C03655=1128.432,274.072,-72.523,-178.249,10.168,149.556
C03656=1128.428,274.321,-72.554,-178.246,10.171,149.556
C03657=1128.424,274.569,-72.583,-178.243,10.173,149.556
C03658=1128.420,274.818,-72.613,-178.240,10.176,149.556
C03659=1128.416,275.065,-72.643,-178.237,10.179,149.556
C03660=1128.412,275.314,-72.672,-178.234,10.181,149.556
C03661=1128.407,275.562,-72.702,-178.231,10.184,149.556
C03662=1128.403,275.810,-72.733,-178.228,10.187,149.555
C03663=1128.399,276.058,-72.762,-178.225,10.189,149.555
C03664=1128.395,276.306,-72.792,-178.221,10.193,149.555
C03665=1128.390,276.554,-72.822,-178.218,10.195,149.555
C03666=1128.386,276.803,-72.852,-178.215,10.198,149.555
C03667=1128.382,277.050,-72.882,-178.212,10.201,149.555
C03668=1128.377,277.299,-72.912,-178.209,10.203,149.554
C03669=1128.374,277.547,-72.943,-178.205,10.207,149.554
C03670=1128.370,277.795,-72.972,-178.202,10.209,149.554
C03671=1128.365,278.043,-73.003,-178.199,10.212,149.554
C03672=1128.361,278.292,-73.032,-178.196,10.214,149.554
C03673=1128.357,278.539,-73.062,-178.192,10.218,149.554
C03674=1128.352,278.788,-73.092,-178.189,10.220,149.553
C03675=1128.348,279.036,-73.123,-178.186,10.223,149.553
C03676=1128.345,279.285,-73.152,-178.182,10.226,149.553
C03677=1128.340,279.532,-73.183,-178.179,10.229,149.553
C03678=1128.336,279.780,-73.213,-178.175,10.231,149.553
C03679=1128.332,279.994,-73.239,-178.172,10.234,149.552
C03680=1128.329,280.207,-73.265,-178.169,10.237,149.552
C03681=1128.325,280.421,-73.291,-178.166,10.239,149.552
C03682=1128.321,280.634,-73.318,-178.163,10.241,149.552
C03683=1128.318,280.848,-73.343,-178.161,10.244,149.552
C03684=1128.314,281.061,-73.370,-178.157,10.246,149.551
C03685=1128.310,281.275,-73.395,-178.154,10.249,149.551
C03686=1128.307,281.489,-73.422,-178.151,10.251,149.551
C03687=1128.303,281.736,-73.452,-178.148,10.254,149.551
C03688=1128.298,281.984,-73.483,-178.145,10.257,149.551
C03689=1128.294,282.233,-73.512,-178.142,10.258,149.550
C03690=1128.290,282.481,-73.543,-178.139,10.261,149.550
C03691=1128.286,282.729,-73.574,-178.136,10.264,149.550
C03692=1128.282,282.977,-73.604,-178.133,10.266,149.550
C03693=1128.277,283.225,-73.634,-178.130,10.269,149.550
C03694=1128.274,283.474,-73.665,-178.127,10.272,149.550
C03695=1128.269,283.722,-73.696,-178.123,10.274,149.549
C03696=1128.265,283.969,-73.726,-178.121,10.277,149.549
C03697=1128.260,284.217,-73.756,-178.117,10.279,149.549
C03698=1128.257,284.466,-73.787,-178.114,10.282,149.549
C03699=1128.253,284.714,-73.818,-178.112,10.284,149.549
C03700=1128.248,284.962,-73.848,-178.109,10.286,149.548
C03701=1128.244,285.209,-73.879,-178.106,10.289,149.548
C03702=1128.240,285.458,-73.909,-178.102,10.292,149.548
C03703=1128.235,285.706,-73.940,-178.099,10.294,149.548
C03704=1128.231,285.954,-73.970,-178.096,10.297,149.548
C03705=1128.227,286.203,-74.001,-178.093,10.299,149.548
C03706=1128.223,286.451,-74.032,-178.090,10.302,149.547
C03707=1128.219,286.698,-74.062,-178.087,10.305,149.547
C03708=1128.215,286.947,-74.093,-178.084,10.307,149.547
C03709=1128.210,287.195,-74.124,-178.081,10.310,149.547
C03710=1128.206,287.443,-74.154,-178.078,10.312,149.547
C03711=1128.203,287.691,-74.186,-178.075,10.314,149.546
C03712=1128.198,287.939,-74.217,-178.072,10.317,149.546
C03713=1128.194,288.186,-74.247,-178.069,10.319,149.546
C03714=1128.190,288.435,-74.278,-178.066,10.322,149.546
C03715=1128.185,288.683,-74.309,-178.062,10.325,149.546
C03716=1128.181,288.931,-74.340,-178.059,10.327,149.546
C03717=1128.178,289.179,-74.370,-178.057,10.330,149.546
C03718=1128.173,289.427,-74.401,-178.053,10.333,149.545
C03719=1128.169,289.675,-74.433,-178.050,10.335,149.545
C03720=1128.165,289.923,-74.463,-178.048,10.337,149.545
C03721=1128.161,290.171,-74.494,-178.045,10.340,149.545
C03722=1128.157,290.419,-74.525,-178.041,10.342,149.545
C03723=1128.152,290.667,-74.556,-178.038,10.345,149.544
C03724=1128.148,290.915,-74.587,-178.035,10.347,149.544
C03725=1128.144,291.163,-74.618,-178.032,10.350,149.544
C03726=1128.141,291.412,-74.649,-178.029,10.353,149.544
C03727=1128.136,291.659,-74.680,-178.026,10.355,149.544
C03728=1128.132,291.907,-74.711,-178.022,10.358,149.543
C03729=1128.128,292.156,-74.742,-178.020,10.360,149.543
C03730=1128.123,292.403,-74.774,-178.017,10.363,149.543
C03731=1128.119,292.652,-74.805,-178.013,10.366,149.543
C03732=1128.115,292.900,-74.835,-178.011,10.368,149.543
C03733=1128.112,293.147,-74.867,-178.008,10.370,149.543
C03734=1128.107,293.395,-74.897,-178.005,10.373,149.543
C03735=1128.104,293.609,-74.924,-178.001,10.375,149.542
C03736=1128.100,293.822,-74.951,-177.999,10.377,149.542
C03737=1128.097,294.035,-74.978,-177.997,10.379,149.542
C03738=1128.093,294.249,-75.005,-177.994,10.382,149.542
C03739=1128.089,294.462,-75.032,-177.991,10.384,149.542
C03740=1128.086,294.676,-75.059,-177.989,10.386,149.542
C03741=1128.082,294.889,-75.086,-177.986,10.388,149.541
C03742=1128.079,295.103,-75.113,-177.983,10.390,149.541
C03743=1128.074,295.350,-75.143,-177.980,10.393,149.541
C03744=1128.070,295.599,-75.175,-177.977,10.395,149.541
C03745=1128.066,295.846,-75.206,-177.974,10.398,149.541
C03746=1128.062,296.095,-75.238,-177.971,10.401,149.541
C03747=1128.058,296.343,-75.270,-177.968,10.403,149.540
C03748=1128.054,296.591,-75.300,-177.965,10.406,149.540
C03749=1128.050,296.839,-75.332,-177.961,10.408,149.540
C03750=1128.045,297.086,-75.363,-177.958,10.411,149.540
C03751=1128.042,297.335,-75.395,-177.956,10.413,149.540
C03752=1128.037,297.582,-75.426,-177.953,10.416,149.540
C03753=1128.033,297.831,-75.458,-177.949,10.418,149.539
C03754=1128.029,298.078,-75.489,-177.947,10.421,149.539
C03755=1128.025,298.327,-75.520,-177.943,10.423,149.539
C03756=1128.021,298.575,-75.553,-177.940,10.426,149.539
C03757=1128.016,298.822,-75.584,-177.937,10.428,149.539
C03758=1128.013,299.070,-75.616,-177.934,10.431,149.538
C03759=1128.008,299.318,-75.647,-177.931,10.434,149.538
C03760=1128.004,299.566,-75.679,-177.928,10.436,149.538
C03761=1128.001,299.814,-75.710,-177.924,10.439,149.538
C03762=1127.996,300.062,-75.742,-177.921,10.441,149.538
C03763=1127.992,300.310,-75.773,-177.918,10.444,149.537
C03764=1127.987,300.558,-75.805,-177.915,10.446,149.537
C03765=1127.984,300.806,-75.837,-177.913,10.448,149.537
C03766=1127.980,301.054,-75.869,-177.909,10.451,149.537
C03767=1127.976,301.301,-75.900,-177.906,10.454,149.537
C03768=1127.971,301.550,-75.931,-177.903,10.456,149.537
C03769=1127.967,301.798,-75.964,-177.900,10.459,149.536
C03770=1127.963,302.046,-75.995,-177.897,10.461,149.536
C03771=1127.959,302.294,-76.027,-177.894,10.464,149.536
C03772=1127.955,302.541,-76.059,-177.890,10.466,149.536
C03773=1127.950,302.789,-76.091,-177.887,10.469,149.536
C03774=1127.947,303.037,-76.123,-177.884,10.472,149.535
C03775=1127.942,303.285,-76.154,-177.881,10.474,149.535
C03776=1127.939,303.533,-76.186,-177.878,10.477,149.535
C03777=1127.934,303.781,-76.219,-177.876,10.479,149.535
C03778=1127.930,304.029,-76.250,-177.872,10.481,149.535
C03779=1127.926,304.277,-76.282,-177.869,10.484,149.535
C03780=1127.922,304.525,-76.314,-177.866,10.486,149.534
C03781=1127.918,304.773,-76.346,-177.863,10.489,149.534
C03782=1127.914,305.020,-76.378,-177.860,10.492,149.534
C03783=1127.909,305.269,-76.410,-177.856,10.494,149.534
C03784=1127.906,305.517,-76.442,-177.853,10.497,149.534
C03785=1127.902,305.765,-76.474,-177.850,10.499,149.533
C03786=1127.897,306.012,-76.506,-177.847,10.502,149.533
C03787=1127.893,306.260,-76.538,-177.844,10.504,149.533
C03788=1127.889,306.508,-76.570,-177.841,10.507,149.533
C03789=1127.885,306.757,-76.602,-177.838,10.510,149.533
C03790=1127.881,307.004,-76.634,-177.835,10.512,149.533
C03791=1127.877,307.217,-76.661,-177.832,10.514,149.532
C03792=1127.874,307.431,-76.689,-177.830,10.516,149.532
C03793=1127.871,307.644,-76.717,-177.826,10.519,149.532
C03794=1127.866,307.857,-76.745,-177.824,10.521,149.532
C03795=1127.863,308.070,-76.772,-177.822,10.523,149.532
C03796=1127.860,308.283,-76.800,-177.818,10.525,149.532
C03797=1127.856,308.497,-76.828,-177.816,10.527,149.531
C03798=1127.853,308.710,-76.856,-177.813,10.530,149.531
C03799=1127.848,308.958,-76.888,-177.810,10.532,149.531
C03800=1127.845,309.205,-76.920,-177.808,10.534,149.531
C03801=1127.840,309.453,-76.953,-177.804,10.537,149.531
C03802=1127.836,309.701,-76.984,-177.801,10.539,149.531
C03803=1127.832,309.950,-77.017,-177.798,10.542,149.530
C03804=1127.829,310.197,-77.049,-177.795,10.544,149.530
C03805=1127.824,310.445,-77.082,-177.792,10.547,149.530
C03806=1127.820,310.692,-77.114,-177.788,10.549,149.530
C03807=1127.816,310.941,-77.147,-177.785,10.552,149.530
C03808=1127.812,311.189,-77.178,-177.782,10.555,149.530
C03809=1127.808,311.436,-77.212,-177.779,10.557,149.529
C03810=1127.804,311.684,-77.243,-177.776,10.560,149.529
C03811=1127.800,311.932,-77.277,-177.772,10.562,149.529
C03812=1127.796,312.179,-77.308,-177.770,10.565,149.529
C03813=1127.792,312.427,-77.341,-177.766,10.567,149.529
C03814=1127.787,312.676,-77.374,-177.763,10.570,149.529
C03815=1127.784,312.923,-77.406,-177.761,10.572,149.528
C03816=1127.779,313.171,-77.439,-177.757,10.574,149.528
C03817=1127.776,313.419,-77.471,-177.754,10.577,149.528
C03818=1127.771,313.667,-77.504,-177.751,10.580,149.528
C03819=1127.767,313.915,-77.537,-177.748,10.582,149.528
C03820=1127.764,314.163,-77.569,-177.745,10.585,149.527
C03821=1127.759,314.411,-77.602,-177.741,10.587,149.527
C03822=1127.754,314.658,-77.634,-177.739,10.590,149.527
C03823=1127.751,314.906,-77.666,-177.735,10.592,149.527
C03824=1127.747,315.153,-77.700,-177.732,10.595,149.526
C03825=1127.742,315.402,-77.732,-177.729,10.598,149.526
C03826=1127.739,315.649,-77.765,-177.726,10.600,149.526
C03827=1127.735,315.897,-77.798,-177.723,10.603,149.526
C03828=1127.730,316.145,-77.830,-177.719,10.605,149.526
C03829=1127.727,316.393,-77.863,-177.716,10.608,149.526
C03830=1127.723,316.640,-77.896,-177.713,10.611,149.525
C03831=1127.718,316.889,-77.928,-177.710,10.612,149.525
C03832=1127.714,317.136,-77.961,-177.707,10.615,149.525
C03833=1127.711,317.384,-77.994,-177.704,10.617,149.525
C03834=1127.707,317.632,-78.027,-177.701,10.620,149.525
C03835=1127.702,317.880,-78.060,-177.698,10.623,149.525
C03836=1127.698,318.128,-78.093,-177.695,10.625,149.524
C03837=1127.694,318.375,-78.126,-177.691,10.627,149.524
C03838=1127.691,318.623,-78.159,-177.688,10.630,149.524
C03839=1127.687,318.871,-78.192,-177.685,10.633,149.524
C03840=1127.682,319.118,-78.225,-177.682,10.635,149.524
C03841=1127.678,319.367,-78.257,-177.679,10.638,149.523
C03842=1127.674,319.614,-78.290,-177.675,10.640,149.523
C03843=1127.670,319.862,-78.323,-177.672,10.643,149.523
C03844=1127.667,320.110,-78.357,-177.669,10.646,149.523
C03845=1127.663,320.358,-78.390,-177.666,10.648,149.523
C03846=1127.659,320.606,-78.423,-177.663,10.651,149.523
C03847=1127.655,320.819,-78.452,-177.660,10.652,149.522
C03848=1127.652,321.032,-78.479,-177.658,10.654,149.522
C03849=1127.648,321.245,-78.508,-177.655,10.657,149.522
C03850=1127.645,321.458,-78.536,-177.652,10.659,149.522
C03851=1127.641,321.671,-78.565,-177.649,10.662,149.522
C03852=1127.638,321.884,-78.594,-177.647,10.663,149.521
C03853=1127.635,322.097,-78.622,-177.644,10.665,149.521
C03854=1127.631,322.310,-78.651,-177.641,10.668,149.521
C03855=1127.627,322.558,-78.684,-177.638,10.671,149.521
C03856=1127.623,322.805,-78.717,-177.635,10.673,149.521
C03857=1127.619,323.053,-78.750,-177.631,10.675,149.521
C03858=1127.614,323.301,-78.783,-177.629,10.677,149.520
C03859=1127.611,323.549,-78.817,-177.626,10.680,149.520
C03860=1127.607,323.796,-78.851,-177.623,10.682,149.520
C03861=1127.603,324.044,-78.884,-177.620,10.685,149.520
C03862=1127.599,324.292,-78.917,-177.616,10.688,149.520
C03863=1127.595,324.540,-78.950,-177.613,10.690,149.519
C03864=1127.591,324.787,-78.983,-177.610,10.693,149.519
C03865=1127.586,325.035,-79.016,-177.607,10.695,149.519
C03866=1127.583,325.283,-79.051,-177.603,10.698,149.519
C03867=1127.579,325.531,-79.084,-177.600,10.700,149.519
C03868=1127.575,325.778,-79.117,-177.597,10.703,149.519
C03869=1127.571,326.026,-79.150,-177.594,10.705,149.518
C03870=1127.567,326.273,-79.184,-177.590,10.708,149.518
C03871=1127.563,326.521,-79.217,-177.588,10.711,149.518
C03872=1127.559,326.769,-79.251,-177.584,10.713,149.518
C03873=1127.555,327.016,-79.284,-177.581,10.715,149.517
C03874=1127.551,327.264,-79.318,-177.578,10.718,149.517
C03875=1127.546,327.512,-79.351,-177.575,10.721,149.517
C03876=1127.543,327.760,-79.386,-177.571,10.723,149.517
C03877=1127.539,328.008,-79.419,-177.569,10.725,149.517
C03878=1127.535,328.255,-79.452,-177.566,10.728,149.517
C03879=1127.531,328.503,-79.486,-177.562,10.730,149.516
C03880=1127.527,328.750,-79.519,-177.559,10.733,149.516
C03881=1127.523,328.999,-79.552,-177.556,10.735,149.516
C03882=1127.519,329.246,-79.587,-177.553,10.738,149.516
C03883=1127.515,329.494,-79.620,-177.550,10.740,149.516
C03884=1127.511,329.741,-79.654,-177.547,10.743,149.515
C03885=1127.507,329.989,-79.688,-177.543,10.745,149.515
C03886=1127.503,330.237,-79.722,-177.540,10.748,149.515
C03887=1127.499,330.485,-79.755,-177.537,10.750,149.515
C03888=1127.495,330.732,-79.789,-177.534,10.753,149.515
C03889=1127.491,330.980,-79.823,-177.530,10.755,149.514
C03890=1127.487,331.227,-79.856,-177.527,10.758,149.514
C03891=1127.483,331.475,-79.890,-177.524,10.761,149.514
C03892=1127.479,331.723,-79.924,-177.521,10.763,149.514
C03893=1127.475,331.970,-79.958,-177.518,10.766,149.514
C03894=1127.471,332.218,-79.992,-177.514,10.768,149.513
C03895=1127.467,332.466,-80.026,-177.511,10.771,149.513
C03896=1127.464,332.713,-80.060,-177.508,10.773,149.513
C03897=1127.459,332.961,-80.093,-177.505,10.775,149.513
C03898=1127.455,333.209,-80.128,-177.502,10.777,149.513
C03899=1127.452,333.456,-80.162,-177.499,10.780,149.513
C03900=1127.447,333.704,-80.195,-177.496,10.783,149.512
C03901=1127.443,333.952,-80.230,-177.492,10.785,149.512
C03902=1127.440,334.199,-80.264,-177.489,10.788,149.512
C03903=1127.436,334.412,-80.293,-177.486,10.790,149.512
C03904=1127.433,334.626,-80.322,-177.483,10.792,149.512
C03905=1127.429,334.838,-80.352,-177.481,10.794,149.511
C03906=1127.426,335.051,-80.381,-177.478,10.796,149.511
C03907=1127.422,335.264,-80.410,-177.476,10.798,149.511
C03908=1127.420,335.477,-80.440,-177.472,10.801,149.511
C03909=1127.416,335.690,-80.469,-177.470,10.803,149.511
C03910=1127.412,335.903,-80.498,-177.467,10.805,149.511
C03911=1127.408,336.150,-80.532,-177.464,10.807,149.510
C03912=1127.405,336.398,-80.566,-177.461,10.810,149.510
C03913=1127.400,336.645,-80.601,-177.458,10.812,149.510
C03914=1127.397,336.893,-80.635,-177.454,10.815,149.510
C03915=1127.392,337.140,-80.670,-177.451,10.817,149.509
C03916=1127.389,337.389,-80.703,-177.448,10.820,149.509
C03917=1127.384,337.636,-80.738,-177.445,10.822,149.509
C03918=1127.380,337.883,-80.771,-177.442,10.825,149.509
C03919=1127.376,338.132,-80.806,-177.438,10.827,149.509
C03920=1127.373,338.379,-80.840,-177.435,10.830,149.509
C03921=1127.369,338.627,-80.875,-177.432,10.833,149.508
C03922=1127.365,338.874,-80.909,-177.429,10.835,149.508
C03923=1127.361,339.122,-80.944,-177.425,10.837,149.508
C03924=1127.357,339.369,-80.978,-177.422,10.840,149.508
C03925=1127.353,339.617,-81.012,-177.419,10.843,149.508
C03926=1127.348,339.865,-81.047,-177.416,10.845,149.507
C03927=1127.345,340.112,-81.081,-177.412,10.848,149.507
C03928=1127.341,340.360,-81.116,-177.409,10.850,149.507
C03929=1127.338,340.607,-81.150,-177.406,10.852,149.507
C03930=1127.333,340.854,-81.185,-177.404,10.854,149.507
C03931=1127.329,341.102,-81.219,-177.400,10.857,149.506
C03932=1127.325,341.350,-81.254,-177.397,10.859,149.506
C03933=1127.321,341.598,-81.288,-177.394,10.862,149.506
C03934=1127.317,341.845,-81.323,-177.390,10.864,149.506
C03935=1127.314,342.093,-81.357,-177.387,10.867,149.505
C03936=1127.309,342.340,-81.392,-177.384,10.870,149.505
C03937=1127.305,342.588,-81.427,-177.381,10.872,149.505
C03938=1127.302,342.835,-81.461,-177.377,10.874,149.505
C03939=1127.298,343.083,-81.496,-177.374,10.877,149.505
C03940=1127.293,343.330,-81.531,-177.371,10.879,149.505
C03941=1127.290,343.578,-81.565,-177.368,10.882,149.504
C03942=1127.286,343.825,-81.600,-177.365,10.885,149.504
C03943=1127.282,344.073,-81.635,-177.361,10.887,149.504
C03944=1127.278,344.320,-81.669,-177.358,10.890,149.504
C03945=1127.274,344.568,-81.704,-177.355,10.892,149.504
C03946=1127.270,344.816,-81.739,-177.351,10.894,149.503
C03947=1127.266,345.063,-81.774,-177.348,10.897,149.503
C03948=1127.262,345.311,-81.809,-177.345,10.900,149.503
C03949=1127.258,345.557,-81.843,-177.342,10.902,149.503
C03950=1127.254,345.806,-81.878,-177.338,10.905,149.503
C03951=1127.250,346.054,-81.913,-177.335,10.907,149.502
C03952=1127.246,346.301,-81.948,-177.332,10.910,149.502
C03953=1127.243,346.548,-81.983,-177.329,10.911,149.502
C03954=1127.239,346.795,-82.018,-177.326,10.914,149.502
C03955=1127.235,347.043,-82.053,-177.323,10.916,149.502
C03956=1127.231,347.291,-82.088,-177.320,10.919,149.501
C03957=1127.226,347.538,-82.123,-177.316,10.921,149.501
C03958=1127.223,347.786,-82.158,-177.313,10.924,149.501
C03959=1127.220,347.998,-82.188,-177.310,10.926,149.501
C03960=1127.216,348.211,-82.218,-177.307,10.928,149.501
C03961=1127.213,348.423,-82.248,-177.305,10.930,149.500
C03962=1127.210,348.637,-82.278,-177.302,10.933,149.500
C03963=1127.206,348.849,-82.309,-177.299,10.934,149.500
C03964=1127.203,349.062,-82.339,-177.296,10.937,149.500
C03965=1127.199,349.275,-82.369,-177.293,10.939,149.500
C03966=1127.197,349.488,-82.399,-177.291,10.941,149.499
C03967=1127.193,349.736,-82.434,-177.287,10.944,149.499
C03968=1127.188,349.983,-82.469,-177.284,10.946,149.499
C03969=1127.185,350.230,-82.504,-177.280,10.950,149.499
C03970=1127.181,350.478,-82.539,-177.276,10.952,149.498
C03971=1127.176,350.725,-82.574,-177.273,10.954,149.498
C03972=1127.173,350.973,-82.610,-177.269,10.957,149.498
C03973=1127.169,351.220,-82.645,-177.265,10.960,149.498
C03974=1127.165,351.468,-82.680,-177.262,10.962,149.497
C03975=1127.161,351.715,-82.715,-177.258,10.965,149.497
C03976=1127.157,351.963,-82.751,-177.254,10.968,149.497
C03977=1127.154,352.210,-82.787,-177.251,10.970,149.497
C03978=1127.150,352.458,-82.821,-177.248,10.973,149.497
C03979=1127.145,352.705,-82.857,-177.243,10.976,149.496
C03980=1127.142,352.952,-82.892,-177.240,10.978,149.496
C03981=1127.138,353.200,-82.928,-177.237,10.980,149.496
C03982=1127.134,353.448,-82.963,-177.233,10.983,149.495
C03983=1127.131,353.695,-82.999,-177.229,10.986,149.495
C03984=1127.126,353.942,-83.034,-177.226,10.988,149.495
C03985=1127.123,354.189,-83.069,-177.223,10.991,149.495
C03986=1127.119,354.437,-83.104,-177.219,10.993,149.494
C03987=1127.114,354.685,-83.140,-177.215,10.996,149.494
C03988=1127.111,354.933,-83.176,-177.212,10.999,149.494
C03989=1127.106,355.180,-83.211,-177.208,11.001,149.494
C03990=1127.103,355.427,-83.247,-177.205,11.004,149.493
C03991=1127.099,355.675,-83.282,-177.201,11.006,149.493
C03992=1127.095,355.922,-83.318,-177.198,11.008,149.493
C03993=1127.092,356.170,-83.353,-177.194,11.011,149.493
C03994=1127.088,356.417,-83.390,-177.191,11.014,149.492
C03995=1127.084,356.664,-83.426,-177.187,11.016,149.492
C03996=1127.080,356.911,-83.461,-177.184,11.018,149.492
C03997=1127.076,357.159,-83.496,-177.180,11.021,149.491
C03998=1127.072,357.406,-83.532,-177.177,11.023,149.491
C03999=1127.069,357.654,-83.568,-177.173,11.025,149.491
C04000=1127.064,357.901,-83.604,-177.170,11.028,149.491
C04001=1127.061,358.149,-83.639,-177.166,11.031,149.490
C04002=1127.057,358.396,-83.676,-177.162,11.033,149.490
C04003=1127.054,358.643,-83.711,-177.159,11.036,149.490
C04004=1127.049,358.891,-83.747,-177.156,11.038,149.490
C04005=1127.046,359.139,-83.783,-177.153,11.041,149.489
C04006=1127.042,359.386,-83.818,-177.149,11.043,149.489
C04007=1127.038,359.632,-83.854,-177.145,11.045,149.489
C04008=1127.034,359.880,-83.890,-177.142,11.048,149.489
C04009=1127.030,360.128,-83.926,-177.139,11.050,149.488
C04010=1127.027,360.374,-83.962,-177.135,11.052,149.488
C04011=1127.022,360.622,-83.998,-177.132,11.055,149.488
C04012=1127.018,360.870,-84.034,-177.129,11.057,149.488
C04013=1127.015,361.117,-84.070,-177.125,11.060,149.487
C04014=1127.011,361.364,-84.106,-177.122,11.062,149.487
C04015=1127.008,361.577,-84.138,-177.119,11.064,149.487
C04016=1127.004,361.790,-84.168,-177.116,11.066,149.487
C04017=1127.001,362.002,-84.199,-177.113,11.068,149.486
C04018=1126.998,362.215,-84.230,-177.110,11.071,149.486
C04019=1126.995,362.428,-84.262,-177.107,11.072,149.486
C04020=1126.992,362.640,-84.293,-177.104,11.075,149.486
C04021=1126.988,362.853,-84.323,-177.101,11.076,149.485
C04022=1126.985,363.065,-84.354,-177.099,11.078,149.485
C04023=1126.981,363.312,-84.391,-177.095,11.081,149.485
C04024=1126.978,363.560,-84.426,-177.092,11.083,149.485
C04025=1126.973,363.807,-84.463,-177.089,11.086,149.485
C04026=1126.970,364.055,-84.499,-177.085,11.088,149.484
C04027=1126.966,364.302,-84.535,-177.082,11.090,149.484
C04028=1126.962,364.549,-84.571,-177.078,11.093,149.484
C04029=1126.958,364.796,-84.608,-177.075,11.095,149.483
C04030=1126.955,365.045,-84.644,-177.072,11.098,149.483
C04031=1126.951,365.292,-84.681,-177.069,11.100,149.483
C04032=1126.947,365.539,-84.717,-177.065,11.103,149.483
C04033=1126.943,365.786,-84.753,-177.062,11.104,149.482
C04034=1126.940,366.033,-84.789,-177.059,11.106,149.482
C04035=1126.936,366.281,-84.826,-177.056,11.109,149.482
C04036=1126.932,366.528,-84.862,-177.052,11.111,149.482
C04037=1126.928,366.775,-84.899,-177.049,11.114,149.482
C04038=1126.924,367.022,-84.935,-177.046,11.116,149.481
C04039=1126.920,367.270,-84.971,-177.042,11.119,149.481
C04040=1126.917,367.517,-85.007,-177.039,11.121,149.481
C04041=1126.913,367.764,-85.044,-177.036,11.123,149.481
C04042=1126.909,368.012,-85.081,-177.033,11.125,149.480
C04043=1126.905,368.259,-85.117,-177.030,11.128,149.480
C04044=1126.901,368.507,-85.154,-177.026,11.130,149.480
C04045=1126.898,368.753,-85.190,-177.023,11.132,149.480
C04046=1126.894,369.001,-85.227,-177.019,11.135,149.479
C04047=1126.890,369.248,-85.264,-177.017,11.137,149.479
C04048=1126.886,369.495,-85.299,-177.014,11.139,149.479
C04049=1126.882,369.743,-85.336,-177.010,11.142,149.479
C04050=1126.879,369.990,-85.373,-177.007,11.144,149.479
C04051=1126.875,370.237,-85.410,-177.004,11.147,149.478
C04052=1126.871,370.485,-85.446,-177.001,11.148,149.478
C04053=1126.867,370.732,-85.483,-176.998,11.151,149.478
C04054=1126.864,370.979,-85.520,-176.994,11.153,149.478
C04055=1126.860,371.226,-85.557,-176.991,11.156,149.478
C04056=1126.856,371.474,-85.594,-176.989,11.158,149.477
C04057=1126.853,371.721,-85.630,-176.985,11.160,149.477
C04058=1126.849,371.968,-85.667,-176.982,11.163,149.477
C04059=1126.845,372.215,-85.704,-176.979,11.165,149.477
C04060=1126.841,372.463,-85.741,-176.976,11.168,149.477
C04061=1126.838,372.710,-85.777,-176.973,11.169,149.476
C04062=1126.834,372.957,-85.814,-176.970,11.172,149.476
C04063=1126.829,373.204,-85.851,-176.966,11.174,149.476
C04064=1126.825,373.451,-85.888,-176.963,11.177,149.476
C04065=1126.823,373.699,-85.924,-176.961,11.179,149.476
C04066=1126.819,373.946,-85.961,-176.957,11.181,149.475
C04067=1126.814,374.193,-85.998,-176.954,11.184,149.475
C04068=1126.810,374.440,-86.035,-176.951,11.185,149.475
C04069=1126.807,374.688,-86.072,-176.949,11.188,149.475
C04070=1126.804,374.935,-86.109,-176.945,11.191,149.475
C04071=1126.800,375.148,-86.141,-176.943,11.192,149.475
C04072=1126.797,375.360,-86.172,-176.940,11.194,149.474
C04073=1126.793,375.573,-86.205,-176.938,11.196,149.474
C04074=1126.790,375.785,-86.236,-176.935,11.199,149.474
C04075=1126.788,375.997,-86.268,-176.932,11.201,149.474
C04076=1126.784,376.210,-86.300,-176.930,11.203,149.474
C04077=1126.781,376.422,-86.332,-176.928,11.205,149.474
C04078=1126.777,376.634,-86.363,-176.925,11.206,149.474
C04079=1126.774,376.882,-86.400,-176.922,11.209,149.473
C04080=1126.770,377.129,-86.438,-176.919,11.212,149.473
C04081=1126.766,377.376,-86.474,-176.916,11.213,149.473
C04082=1126.763,377.624,-86.512,-176.913,11.216,149.473
C04083=1126.759,377.870,-86.549,-176.910,11.219,149.473
C04084=1126.755,378.117,-86.586,-176.907,11.220,149.473
C04085=1126.751,378.365,-86.623,-176.904,11.223,149.473
C04086=1126.748,378.612,-86.661,-176.901,11.226,149.472
C04087=1126.743,378.859,-86.698,-176.899,11.228,149.472
C04088=1126.740,379.107,-86.735,-176.895,11.230,149.472
C04089=1126.736,379.354,-86.773,-176.892,11.233,149.472
C04090=1126.732,379.601,-86.809,-176.890,11.235,149.472
C04091=1126.729,379.848,-86.847,-176.887,11.237,149.472
C04092=1126.725,380.095,-86.884,-176.884,11.240,149.472
C04093=1126.721,380.342,-86.921,-176.881,11.242,149.472
C04094=1126.717,380.590,-86.959,-176.878,11.245,149.472
C04095=1126.713,380.837,-86.996,-176.875,11.247,149.472
C04096=1126.710,381.084,-87.034,-176.873,11.249,149.471
C04097=1126.706,381.331,-87.071,-176.870,11.252,149.471
C04098=1126.702,381.578,-87.108,-176.867,11.254,149.471
C04099=1126.699,381.826,-87.146,-176.864,11.257,149.471
C04100=1126.695,382.072,-87.183,-176.862,11.259,149.471
C04101=1126.692,382.320,-87.220,-176.859,11.261,149.471
C04102=1126.688,382.567,-87.258,-176.856,11.264,149.471
C04103=1126.684,382.813,-87.295,-176.853,11.267,149.471
C04104=1126.680,383.061,-87.333,-176.851,11.269,149.471
C04105=1126.677,383.308,-87.370,-176.847,11.271,149.471
C04106=1126.673,383.556,-87.407,-176.846,11.274,149.471
C04107=1126.669,383.803,-87.446,-176.844,11.275,149.471
C04108=1126.665,384.049,-87.483,-176.842,11.277,149.471
C04109=1126.661,384.297,-87.520,-176.841,11.279,149.471
C04110=1126.658,384.544,-87.558,-176.839,11.281,149.471
C04111=1126.654,384.791,-87.596,-176.838,11.283,149.471
C04112=1126.650,385.038,-87.633,-176.836,11.284,149.471
C04113=1126.647,385.285,-87.671,-176.835,11.287,149.471
C04114=1126.643,385.532,-87.708,-176.833,11.288,149.471
C04115=1126.639,385.780,-87.746,-176.831,11.291,149.472
C04116=1126.635,386.027,-87.784,-176.830,11.292,149.472
C04117=1126.632,386.274,-87.822,-176.828,11.295,149.472
C04118=1126.628,386.521,-87.859,-176.827,11.296,149.472
C04119=1126.625,386.768,-87.896,-176.825,11.299,149.472
C04120=1126.621,387.015,-87.934,-176.824,11.300,149.472
C04121=1126.617,387.262,-87.972,-176.822,11.303,149.472
C04122=1126.613,387.510,-88.009,-176.821,11.304,149.473
C04123=1126.609,387.756,-88.047,-176.820,11.307,149.473
C04124=1126.606,388.004,-88.085,-176.818,11.309,149.473
C04125=1126.602,388.250,-88.123,-176.817,11.311,149.473
C04126=1126.599,388.498,-88.160,-176.816,11.313,149.473
C04127=1126.595,388.710,-88.192,-176.815,11.315,149.474
C04128=1126.592,388.923,-88.225,-176.813,11.317,149.474
C04129=1126.589,389.135,-88.257,-176.812,11.319,149.474
C04130=1126.586,389.347,-88.289,-176.811,11.321,149.474
C04131=1126.582,389.560,-88.322,-176.810,11.322,149.474
C04132=1126.580,389.772,-88.354,-176.809,11.324,149.475
C04133=1126.577,389.985,-88.387,-176.808,11.326,149.475
C04134=1126.573,390.197,-88.420,-176.806,11.329,149.475
C04135=1126.569,390.443,-88.457,-176.806,11.331,149.475
C04136=1126.566,390.691,-88.495,-176.804,11.333,149.476
C04137=1126.562,390.937,-88.533,-176.803,11.335,149.476
C04138=1126.558,391.185,-88.571,-176.802,11.338,149.476
C04139=1126.555,391.431,-88.609,-176.800,11.341,149.477
C04140=1126.551,391.679,-88.647,-176.799,11.342,149.477
C04141=1126.548,391.926,-88.685,-176.798,11.345,149.477
C04142=1126.544,392.173,-88.723,-176.797,11.347,149.477
C04143=1126.540,392.421,-88.760,-176.796,11.350,149.478
C04144=1126.536,392.667,-88.798,-176.795,11.353,149.478
C04145=1126.532,392.915,-88.836,-176.794,11.355,149.479
C04146=1126.529,393.162,-88.874,-176.793,11.358,149.479
C04147=1126.525,393.409,-88.912,-176.792,11.360,149.479
C04148=1126.522,393.655,-88.949,-176.791,11.363,149.480
C04149=1126.518,393.903,-88.988,-176.789,11.365,149.480
C04150=1126.514,394.150,-89.025,-176.789,11.367,149.481
C04151=1126.511,394.397,-89.063,-176.787,11.370,149.481
C04152=1126.507,394.644,-89.102,-176.786,11.373,149.481
C04153=1126.503,394.891,-89.139,-176.786,11.375,149.482
C04154=1126.500,395.138,-89.177,-176.785,11.378,149.482
C04155=1126.495,395.385,-89.216,-176.784,11.381,149.483
C04156=1126.492,395.632,-89.253,-176.782,11.384,149.483
C04157=1126.488,395.879,-89.291,-176.782,11.386,149.484
C04158=1126.484,396.127,-89.330,-176.780,11.389,149.484
C04159=1126.481,396.374,-89.368,-176.780,11.393,149.485
C04160=1126.477,396.620,-89.405,-176.779,11.395,149.485
C04161=1126.474,396.868,-89.444,-176.778,11.398,149.486
C04162=1126.470,397.114,-89.481,-176.777,11.401,149.486
C04163=1126.466,397.362,-89.520,-176.776,11.404,149.487
C04164=1126.463,397.609,-89.558,-176.776,11.406,149.488
C04165=1126.459,397.856,-89.595,-176.775,11.410,149.488
C04166=1126.455,398.103,-89.635,-176.774,11.413,149.489
C04167=1126.451,398.349,-89.672,-176.773,11.416,149.489
C04168=1126.448,398.597,-89.710,-176.772,11.419,149.490
C04169=1126.444,398.844,-89.749,-176.772,11.421,149.490
C04170=1126.441,399.091,-89.786,-176.771,11.425,149.491
C04171=1126.437,399.338,-89.825,-176.771,11.428,149.492
C04172=1126.433,399.585,-89.862,-176.769,11.431,149.492
C04173=1126.430,399.832,-89.900,-176.769,11.434,149.493
C04174=1126.426,400.079,-89.939,-176.768,11.438,149.494
C04175=1126.422,400.326,-89.977,-176.767,11.441,149.494
C04176=1126.418,400.573,-90.016,-176.767,11.444,149.495
C04177=1126.415,400.821,-90.053,-176.767,11.447,149.496
C04178=1126.411,401.068,-90.092,-176.766,11.450,149.496
C04179=1126.407,401.315,-90.130,-176.766,11.454,149.497
C04180=1126.405,401.561,-90.168,-176.765,11.457,149.498
C04181=1126.400,401.808,-90.206,-176.764,11.461,149.499
C04182=1126.397,402.056,-90.244,-176.764,11.464,149.500
C04183=1126.393,402.268,-90.277,-176.763,11.467,149.500
C04184=1126.390,402.480,-90.310,-176.763,11.470,149.501
C04185=1126.387,402.692,-90.343,-176.763,11.473,149.502
C04186=1126.384,402.904,-90.376,-176.762,11.476,149.502
C04187=1126.381,403.117,-90.409,-176.762,11.480,149.503
C04188=1126.377,403.329,-90.442,-176.762,11.482,149.504
C04189=1126.374,403.541,-90.475,-176.761,11.485,149.504
C04190=1126.371,403.753,-90.507,-176.761,11.488,149.505
C04191=1126.368,404.000,-90.546,-176.760,11.492,149.506
C04192=1126.364,404.247,-90.584,-176.760,11.495,149.507
C04193=1126.361,404.495,-90.623,-176.760,11.499,149.508
C04194=1126.357,404.741,-90.660,-176.759,11.503,149.508
C04195=1126.353,404.988,-90.699,-176.759,11.506,149.509
C04196=1126.350,405.236,-90.737,-176.759,11.510,149.510
C04197=1126.345,405.482,-90.776,-176.758,11.515,149.511
C04198=1126.343,405.729,-90.814,-176.758,11.518,149.512
C04199=1126.339,405.977,-90.853,-176.758,11.522,149.513
C04200=1126.335,406.223,-90.890,-176.758,11.526,149.514
C04201=1126.331,406.470,-90.930,-176.757,11.530,149.515
C04202=1126.328,406.717,-90.968,-176.758,11.534,149.516
C04203=1126.323,406.964,-91.006,-176.757,11.537,149.517
C04204=1126.320,407.211,-91.045,-176.757,11.541,149.518
C04205=1126.317,407.459,-91.083,-176.757,11.545,149.519
C04206=1126.313,407.705,-91.122,-176.757,11.550,149.520
C04207=1126.309,407.952,-91.160,-176.757,11.554,149.521
C04208=1126.305,408.200,-91.198,-176.757,11.558,149.522
C04209=1126.302,408.446,-91.237,-176.757,11.562,149.523
C04210=1126.299,408.694,-91.275,-176.757,11.566,149.524
C04211=1126.295,408.940,-91.314,-176.757,11.571,149.525
C04212=1126.291,409.187,-91.352,-176.757,11.575,149.526
C04213=1126.288,409.434,-91.392,-176.757,11.579,149.528
C04214=1126.284,409.681,-91.429,-176.757,11.583,149.529
C04215=1126.280,409.929,-91.468,-176.757,11.588,149.530
C04216=1126.277,410.175,-91.506,-176.757,11.592,149.531
C04217=1126.273,410.423,-91.545,-176.757,11.596,149.532
C04218=1126.269,410.669,-91.584,-176.757,11.601,149.533
C04219=1126.266,410.916,-91.622,-176.757,11.605,149.535
C04220=1126.262,411.163,-91.661,-176.757,11.610,149.536
C04221=1126.259,411.411,-91.699,-176.757,11.615,149.537
C04222=1126.255,411.657,-91.738,-176.758,11.619,149.538
C04223=1126.251,411.904,-91.776,-176.758,11.623,149.540
C04224=1126.248,412.151,-91.815,-176.758,11.629,149.541
C04225=1126.244,412.398,-91.854,-176.758,11.633,149.542
C04226=1126.240,412.646,-91.893,-176.758,11.638,149.543
C04227=1126.237,412.891,-91.931,-176.759,11.643,149.545
C04228=1126.233,413.139,-91.970,-176.760,11.647,149.546
C04229=1126.229,413.386,-92.009,-176.759,11.652,149.547
C04230=1126.226,413.633,-92.047,-176.760,11.657,149.549
C04231=1126.222,413.880,-92.086,-176.760,11.662,149.550
C04232=1126.219,414.126,-92.124,-176.761,11.666,149.551
C04233=1126.216,414.374,-92.163,-176.761,11.672,149.553
C04234=1126.213,414.621,-92.201,-176.762,11.676,149.554
C04235=1126.212,414.868,-92.240,-176.762,11.682,149.556
C04236=1126.212,415.115,-92.278,-176.763,11.687,149.557
C04237=1126.211,415.362,-92.316,-176.763,11.692,149.559
C04238=1126.211,415.609,-92.355,-176.764,11.697,149.560
C04239=1126.211,415.821,-92.387,-176.764,11.701,149.561
C04240=1126.213,416.033,-92.420,-176.765,11.705,149.563
C04241=1126.214,416.245,-92.453,-176.766,11.710,149.564
C04242=1126.216,416.457,-92.486,-176.766,11.714,149.565
C04243=1126.219,416.670,-92.517,-176.767,11.719,149.566
C04244=1126.221,416.881,-92.549,-176.767,11.723,149.568
C04245=1126.224,417.094,-92.582,-176.768,11.728,149.569
C04246=1126.228,417.305,-92.615,-176.769,11.732,149.571
C04247=1125.809,417.305,-92.678,-176.761,11.736,149.570
C04248=1125.806,417.093,-92.645,-176.761,11.732,149.569
C04249=1125.802,416.881,-92.613,-176.760,11.727,149.567
C04250=1125.799,416.668,-92.580,-176.760,11.723,149.566
C04251=1125.797,416.457,-92.548,-176.759,11.719,149.564
C04252=1125.795,416.245,-92.515,-176.758,11.714,149.563
C04253=1125.794,416.033,-92.482,-176.758,11.710,149.562
C04254=1125.792,415.821,-92.450,-176.757,11.705,149.561
C04255=1125.792,415.609,-92.417,-176.757,11.701,149.559
C04256=1125.792,415.362,-92.378,-176.756,11.695,149.558
C04257=1125.792,415.115,-92.340,-176.756,11.691,149.556
C04258=1125.793,414.868,-92.302,-176.755,11.685,149.555
C04259=1125.794,414.621,-92.264,-176.754,11.681,149.554
C04260=1125.797,414.373,-92.225,-176.755,11.676,149.552
C04261=1125.800,414.127,-92.186,-176.754,11.671,149.551
C04262=1125.803,413.880,-92.148,-176.754,11.666,149.549
C04263=1125.806,413.633,-92.109,-176.753,11.661,149.548
C04264=1125.810,413.386,-92.070,-176.753,11.656,149.547
C04265=1125.814,413.139,-92.032,-176.753,11.651,149.545
C04266=1125.817,412.892,-91.993,-176.753,11.646,149.544
C04267=1125.821,412.645,-91.955,-176.753,11.641,149.543
C04268=1125.824,412.398,-91.916,-176.752,11.637,149.541
C04269=1125.828,412.151,-91.877,-176.752,11.632,149.540
C04270=1125.832,411.904,-91.839,-176.752,11.627,149.539
C04271=1125.835,411.657,-91.800,-176.751,11.623,149.538
C04272=1125.839,411.410,-91.761,-176.752,11.618,149.536
C04273=1125.842,411.163,-91.723,-176.751,11.614,149.535
C04274=1125.847,410.916,-91.684,-176.752,11.609,149.534
C04275=1125.850,410.669,-91.645,-176.751,11.604,149.533
C04276=1125.853,410.422,-91.607,-176.751,11.600,149.532
C04277=1125.857,410.175,-91.568,-176.751,11.595,149.530
C04278=1125.861,409.929,-91.530,-176.751,11.591,149.529
C04279=1125.864,409.682,-91.491,-176.751,11.587,149.528
C04280=1125.868,409.434,-91.453,-176.751,11.582,149.527
C04281=1125.871,409.187,-91.414,-176.751,11.578,149.526
C04282=1125.876,408.940,-91.376,-176.751,11.574,149.525
C04283=1125.879,408.694,-91.337,-176.751,11.569,149.524
C04284=1125.883,408.446,-91.299,-176.751,11.565,149.523
C04285=1125.886,408.199,-91.259,-176.751,11.561,149.522
C04286=1125.890,407.953,-91.222,-176.751,11.557,149.520
C04287=1125.894,407.705,-91.183,-176.752,11.553,149.520
C04288=1125.897,407.458,-91.145,-176.752,11.549,149.519
C04289=1125.901,407.211,-91.106,-176.752,11.545,149.517
C04290=1125.904,406.965,-91.068,-176.752,11.541,149.516
C04291=1125.908,406.717,-91.029,-176.752,11.537,149.516
C04292=1125.911,406.470,-90.991,-176.753,11.532,149.514
C04293=1125.916,406.224,-90.952,-176.753,11.529,149.514
C04294=1125.920,405.976,-90.914,-176.753,11.525,149.512
C04295=1125.923,405.729,-90.876,-176.753,11.521,149.512
C04296=1125.926,405.482,-90.837,-176.754,11.517,149.511
C04297=1125.930,405.235,-90.799,-176.754,11.514,149.510
C04298=1125.934,404.988,-90.760,-176.755,11.509,149.509
C04299=1125.937,404.741,-90.722,-176.755,11.506,149.508
C04300=1125.941,404.494,-90.684,-176.755,11.502,149.507
C04301=1125.945,404.247,-90.646,-176.756,11.498,149.506
C04302=1125.948,404.000,-90.607,-176.756,11.495,149.505
C04303=1125.952,403.754,-90.569,-176.756,11.491,149.505
C04304=1125.955,403.541,-90.535,-176.757,11.488,149.504
C04305=1125.958,403.329,-90.503,-176.757,11.485,149.503
C04306=1125.962,403.116,-90.470,-176.758,11.481,149.502
C04307=1125.965,402.905,-90.437,-176.758,11.479,149.502
C04308=1125.968,402.692,-90.404,-176.758,11.475,149.501
C04309=1125.970,402.480,-90.371,-176.759,11.472,149.500
C04310=1125.974,402.268,-90.339,-176.759,11.470,149.500
C04311=1125.977,402.056,-90.306,-176.760,11.466,149.499
C04312=1125.981,401.809,-90.267,-176.760,11.463,149.498
C04313=1125.984,401.562,-90.229,-176.761,11.460,149.498
C04314=1125.988,401.315,-90.191,-176.761,11.456,149.497
C04315=1125.992,401.067,-90.153,-176.762,11.453,149.496
C04316=1125.995,400.821,-90.114,-176.763,11.449,149.495
C04317=1125.999,400.574,-90.076,-176.763,11.447,149.495
C04318=1126.002,400.326,-90.038,-176.764,11.443,149.494
C04319=1126.007,400.079,-90.000,-176.764,11.440,149.493
C04320=1126.010,399.832,-89.962,-176.765,11.437,149.493
C04321=1126.014,399.585,-89.924,-176.766,11.434,149.492
C04322=1126.017,399.339,-89.885,-176.767,11.430,149.491
C04323=1126.020,399.091,-89.847,-176.768,11.427,149.491
C04324=1126.025,398.845,-89.809,-176.769,11.424,149.490
C04325=1126.028,398.597,-89.771,-176.769,11.421,149.490
C04326=1126.032,398.350,-89.732,-176.769,11.418,149.489
C04327=1126.036,398.103,-89.695,-176.771,11.415,149.488
C04328=1126.039,397.856,-89.657,-176.771,11.412,149.488
C04329=1126.044,397.609,-89.619,-176.772,11.409,149.487
C04330=1126.046,397.362,-89.580,-176.773,11.406,149.487
C04331=1126.050,397.115,-89.542,-176.774,11.403,149.486
C04332=1126.054,396.868,-89.504,-176.775,11.400,149.486
C04333=1126.057,396.621,-89.466,-176.776,11.397,149.485
C04334=1126.062,396.374,-89.428,-176.777,11.394,149.484
C04335=1126.065,396.127,-89.390,-176.778,11.391,149.484
C04336=1126.068,395.879,-89.352,-176.779,11.388,149.483
C04337=1126.073,395.633,-89.314,-176.779,11.386,149.483
C04338=1126.076,395.385,-89.276,-176.780,11.383,149.483
C04339=1126.080,395.139,-89.238,-176.782,11.380,149.482
C04340=1126.084,394.891,-89.200,-176.783,11.377,149.482
C04341=1126.087,394.645,-89.162,-176.783,11.375,149.481
C04342=1126.091,394.397,-89.124,-176.785,11.372,149.481
C04343=1126.095,394.150,-89.086,-176.786,11.369,149.480
C04344=1126.098,393.903,-89.048,-176.787,11.367,149.480
C04345=1126.102,393.656,-89.010,-176.788,11.364,149.480
C04346=1126.106,393.409,-88.972,-176.789,11.361,149.479
C04347=1126.109,393.162,-88.934,-176.790,11.359,149.479
C04348=1126.113,392.915,-88.897,-176.791,11.356,149.478
C04349=1126.117,392.668,-88.858,-176.793,11.354,149.478
C04350=1126.121,392.421,-88.820,-176.793,11.352,149.478
C04351=1126.124,392.174,-88.782,-176.794,11.349,149.477
C04352=1126.128,391.927,-88.746,-176.796,11.346,149.477
C04353=1126.132,391.679,-88.707,-176.797,11.344,149.477
C04354=1126.135,391.432,-88.669,-176.798,11.341,149.476
C04355=1126.139,391.185,-88.632,-176.800,11.339,149.476
C04356=1126.142,390.938,-88.594,-176.801,11.337,149.476
C04357=1126.147,390.691,-88.555,-176.802,11.334,149.475
C04358=1126.150,390.444,-88.518,-176.804,11.331,149.475
C04359=1126.154,390.197,-88.480,-176.804,11.330,149.475
C04360=1126.157,389.985,-88.447,-176.806,11.328,149.475
C04361=1126.160,389.773,-88.415,-176.807,11.325,149.474
C04362=1126.163,389.560,-88.382,-176.808,11.323,149.474
C04363=1126.166,389.347,-88.350,-176.809,11.322,149.474
C04364=1126.169,389.135,-88.318,-176.810,11.320,149.474
C04365=1126.172,388.923,-88.285,-176.811,11.318,149.474
C04366=1126.176,388.711,-88.253,-176.813,11.316,149.473
C04367=1126.179,388.499,-88.221,-176.814,11.314,149.473
C04368=1126.183,388.252,-88.183,-176.815,11.312,149.473
C04369=1126.187,388.004,-88.145,-176.817,11.310,149.473
C04370=1126.190,387.757,-88.108,-176.818,11.307,149.473
C04371=1126.194,387.510,-88.070,-176.820,11.306,149.472
C04372=1126.197,387.263,-88.032,-176.821,11.303,149.472
C04373=1126.201,387.016,-87.995,-176.822,11.301,149.472
C04374=1126.205,386.769,-87.957,-176.824,11.299,149.472
C04375=1126.209,386.521,-87.919,-176.825,11.297,149.472
C04376=1126.212,386.275,-87.881,-176.827,11.295,149.472
C04377=1126.216,386.027,-87.844,-176.829,11.293,149.472
C04378=1126.220,385.780,-87.806,-176.830,11.291,149.471
C04379=1126.223,385.533,-87.769,-176.832,11.290,149.471
C04380=1126.227,385.286,-87.732,-176.834,11.287,149.471
C04381=1126.231,385.038,-87.693,-176.835,11.286,149.471
C04382=1126.235,384.792,-87.656,-176.837,11.283,149.471
C04383=1126.238,384.544,-87.618,-176.838,11.282,149.471
C04384=1126.242,384.297,-87.581,-176.840,11.279,149.471
C04385=1126.246,384.051,-87.543,-176.841,11.278,149.471
C04386=1126.249,383.803,-87.506,-176.843,11.276,149.471
C04387=1126.253,383.556,-87.468,-176.845,11.274,149.471
C04388=1126.256,383.309,-87.430,-176.847,11.272,149.471
C04389=1126.261,383.062,-87.393,-176.850,11.269,149.471
C04390=1126.264,382.814,-87.355,-176.852,11.267,149.471
C04391=1126.268,382.567,-87.318,-176.855,11.264,149.471
C04392=1126.272,382.320,-87.281,-176.858,11.262,149.471
C04393=1126.275,382.073,-87.243,-176.860,11.260,149.471
C04394=1126.279,381.826,-87.206,-176.863,11.257,149.471
C04395=1126.283,381.579,-87.168,-176.866,11.255,149.471
C04396=1126.287,381.332,-87.131,-176.869,11.253,149.471
C04397=1126.290,381.085,-87.093,-176.872,11.250,149.471
C04398=1126.294,380.837,-87.056,-176.874,11.248,149.471
C04399=1126.298,380.591,-87.019,-176.877,11.245,149.472
C04400=1126.301,380.343,-86.981,-176.880,11.242,149.472
C04401=1126.305,380.096,-86.944,-176.883,11.241,149.472
C04402=1126.309,379.849,-86.907,-176.886,11.238,149.472
C04403=1126.313,379.601,-86.870,-176.889,11.235,149.472
C04404=1126.316,379.354,-86.832,-176.891,11.233,149.472
C04405=1126.320,379.107,-86.795,-176.895,11.231,149.472
C04406=1126.324,378.860,-86.757,-176.898,11.228,149.472
C04407=1126.328,378.613,-86.721,-176.900,11.226,149.473
C04408=1126.332,378.366,-86.684,-176.903,11.224,149.473
C04409=1126.335,378.118,-86.646,-176.907,11.221,149.473
C04410=1126.339,377.871,-86.609,-176.909,11.219,149.473
C04411=1126.343,377.624,-86.572,-176.912,11.217,149.473
C04412=1126.346,377.377,-86.534,-176.915,11.214,149.473
C04413=1126.350,377.130,-86.498,-176.918,11.212,149.473
C04414=1126.354,376.883,-86.461,-176.921,11.210,149.473
C04415=1126.357,376.635,-86.424,-176.924,11.207,149.473
C04416=1126.361,376.422,-86.391,-176.927,11.205,149.474
C04417=1126.365,376.210,-86.360,-176.929,11.203,149.474
C04418=1126.367,375.998,-86.328,-176.931,11.201,149.474
C04419=1126.371,375.785,-86.296,-176.934,11.199,149.474
C04420=1126.374,375.573,-86.264,-176.937,11.197,149.474
C04421=1126.378,375.360,-86.233,-176.939,11.195,149.474
C04422=1126.380,375.148,-86.201,-176.942,11.193,149.475
C04423=1126.383,374.936,-86.169,-176.944,11.191,149.475
C04424=1126.387,374.689,-86.132,-176.948,11.189,149.475
C04425=1126.391,374.441,-86.095,-176.951,11.186,149.475
C04426=1126.395,374.194,-86.058,-176.954,11.184,149.475
C04427=1126.399,373.947,-86.021,-176.956,11.182,149.475
C04428=1126.402,373.700,-85.985,-176.960,11.179,149.476
C04429=1126.406,373.453,-85.948,-176.963,11.177,149.476
C04430=1126.410,373.205,-85.910,-176.966,11.174,149.476
C04431=1126.414,372.958,-85.874,-176.969,11.173,149.476
C04432=1126.417,372.711,-85.837,-176.972,11.170,149.476
C04433=1126.421,372.464,-85.800,-176.976,11.168,149.477
C04434=1126.425,372.216,-85.763,-176.978,11.165,149.477
C04435=1126.429,371.969,-85.726,-176.981,11.163,149.477
C04436=1126.432,371.722,-85.690,-176.984,11.161,149.477
C04437=1126.436,371.475,-85.653,-176.988,11.158,149.477
C04438=1126.440,371.227,-85.616,-176.991,11.156,149.477
C04439=1126.443,370.980,-85.580,-176.994,11.154,149.478
C04440=1126.447,370.733,-85.543,-176.997,11.151,149.478
C04441=1126.451,370.485,-85.506,-177.000,11.149,149.478
C04442=1126.455,370.238,-85.469,-177.004,11.147,149.478
C04443=1126.459,369.991,-85.433,-177.007,11.144,149.479
C04444=1126.463,369.743,-85.397,-177.010,11.142,149.479
C04445=1126.467,369.496,-85.360,-177.013,11.140,149.479
C04446=1126.470,369.249,-85.323,-177.016,11.137,149.479
C04447=1126.474,369.002,-85.286,-177.019,11.135,149.479
C04448=1126.478,368.755,-85.250,-177.023,11.132,149.480
C04449=1126.482,368.507,-85.213,-177.026,11.130,149.480
C04450=1126.486,368.260,-85.177,-177.029,11.128,149.480
C04451=1126.489,368.013,-85.141,-177.032,11.126,149.480
C04452=1126.493,367.765,-85.104,-177.035,11.123,149.481
C04453=1126.496,367.518,-85.067,-177.039,11.121,149.481
C04454=1126.501,367.270,-85.031,-177.042,11.118,149.481
C04455=1126.505,367.023,-84.994,-177.046,11.116,149.481
C04456=1126.508,366.776,-84.958,-177.048,11.115,149.482
C04457=1126.512,366.529,-84.921,-177.052,11.112,149.482
C04458=1126.516,366.281,-84.886,-177.055,11.110,149.482
C04459=1126.520,366.034,-84.849,-177.058,11.107,149.482
C04460=1126.524,365.787,-84.813,-177.062,11.105,149.482
C04461=1126.528,365.540,-84.776,-177.065,11.102,149.483
C04462=1126.531,365.293,-84.740,-177.068,11.100,149.483
C04463=1126.535,365.045,-84.704,-177.072,11.098,149.483
C04464=1126.538,364.797,-84.667,-177.075,11.095,149.483
C04465=1126.543,364.549,-84.631,-177.078,11.093,149.484
C04466=1126.546,364.303,-84.595,-177.081,11.091,149.484
C04467=1126.550,364.055,-84.558,-177.084,11.088,149.484
C04468=1126.554,363.808,-84.523,-177.088,11.086,149.484
C04469=1126.557,363.561,-84.486,-177.091,11.084,149.485
C04470=1126.561,363.313,-84.450,-177.095,11.081,149.485
C04471=1126.565,363.066,-84.414,-177.098,11.079,149.485
C04472=1126.568,362.853,-84.383,-177.101,11.077,149.485
C04473=1126.572,362.641,-84.352,-177.104,11.075,149.486
C04474=1126.575,362.428,-84.321,-177.107,11.073,149.486
C04475=1126.578,362.216,-84.290,-177.110,11.071,149.486
C04476=1126.582,362.004,-84.259,-177.112,11.069,149.486
C04477=1126.585,361.791,-84.228,-177.116,11.066,149.486
C04478=1126.588,361.578,-84.197,-177.118,11.064,149.487
C04479=1126.591,361.365,-84.166,-177.121,11.063,149.487
C04480=1126.595,361.118,-84.130,-177.124,11.060,149.487
C04481=1126.599,360.871,-84.094,-177.128,11.058,149.488
C04482=1126.602,360.623,-84.058,-177.131,11.056,149.488
C04483=1126.606,360.376,-84.022,-177.135,11.053,149.488
C04484=1126.611,360.129,-83.986,-177.138,11.051,149.488
C04485=1126.614,359.882,-83.950,-177.142,11.048,149.489
C04486=1126.618,359.634,-83.915,-177.145,11.045,149.489
C04487=1126.623,359.386,-83.879,-177.149,11.043,149.489
C04488=1126.626,359.139,-83.842,-177.152,11.040,149.489
C04489=1126.630,358.892,-83.807,-177.156,11.038,149.490
C04490=1126.633,358.644,-83.771,-177.159,11.036,149.490
C04491=1126.638,358.397,-83.735,-177.162,11.033,149.490
C04492=1126.641,358.150,-83.699,-177.166,11.031,149.490
C04493=1126.645,357.902,-83.663,-177.169,11.029,149.491
C04494=1126.648,357.655,-83.628,-177.173,11.026,149.491
C04495=1126.652,357.407,-83.592,-177.176,11.024,149.491
C04496=1126.656,357.159,-83.556,-177.179,11.021,149.491
C04497=1126.661,356.913,-83.521,-177.183,11.019,149.492
C04498=1126.664,356.665,-83.485,-177.187,11.016,149.492
C04499=1126.668,356.418,-83.450,-177.190,11.013,149.492
C04500=1126.672,356.170,-83.414,-177.194,11.011,149.492
C04501=1126.676,355.923,-83.377,-177.197,11.009,149.493
C04502=1126.679,355.675,-83.342,-177.201,11.006,149.493
C04503=1126.683,355.428,-83.306,-177.204,11.004,149.493
C04504=1126.687,355.181,-83.271,-177.208,11.001,149.493
C04505=1126.691,354.934,-83.236,-177.212,10.999,149.494
C04506=1126.695,354.686,-83.200,-177.215,10.996,149.494
C04507=1126.699,354.438,-83.165,-177.218,10.994,149.494
C04508=1126.702,354.190,-83.130,-177.222,10.991,149.494
C04509=1126.706,353.943,-83.094,-177.225,10.989,149.495
C04510=1126.711,353.696,-83.058,-177.229,10.986,149.495
C04511=1126.715,353.448,-83.023,-177.232,10.983,149.495
C04512=1126.718,353.201,-82.987,-177.236,10.981,149.496
C04513=1126.722,352.953,-82.952,-177.239,10.979,149.496
C04514=1126.726,352.707,-82.917,-177.243,10.976,149.496
C04515=1126.730,352.459,-82.881,-177.247,10.973,149.496
C04516=1126.734,352.211,-82.846,-177.250,10.971,149.497
C04517=1126.737,351.963,-82.811,-177.254,10.968,149.497
C04518=1126.741,351.716,-82.775,-177.258,10.965,149.497
C04519=1126.745,351.469,-82.740,-177.261,10.963,149.497
C04520=1126.749,351.221,-82.705,-177.264,10.960,149.498
C04521=1126.753,350.973,-82.670,-177.268,10.957,149.498
C04522=1126.757,350.727,-82.634,-177.272,10.955,149.498
C04523=1126.761,350.479,-82.599,-177.275,10.952,149.498
C04524=1126.765,350.231,-82.564,-177.279,10.949,149.499
C04525=1126.769,349.984,-82.528,-177.283,10.947,149.499
C04526=1126.772,349.737,-82.494,-177.286,10.944,149.499
C04527=1126.776,349.489,-82.459,-177.290,10.941,149.499
C04528=1126.779,349.276,-82.428,-177.292,10.939,149.500
C04529=1126.783,349.063,-82.398,-177.296,10.937,149.500
C04530=1126.787,348.851,-82.369,-177.298,10.935,149.500
C04531=1126.790,348.638,-82.338,-177.301,10.933,149.500
C04532=1126.793,348.425,-82.308,-177.304,10.931,149.500
C04533=1126.796,348.212,-82.278,-177.306,10.929,149.500
C04534=1126.800,347.999,-82.248,-177.310,10.926,149.501
C04535=1126.803,347.787,-82.218,-177.312,10.924,149.501
C04536=1126.807,347.540,-82.183,-177.315,10.922,149.501
C04537=1126.811,347.292,-82.147,-177.319,10.919,149.501
C04538=1126.815,347.044,-82.112,-177.322,10.917,149.501
C04539=1126.819,346.797,-82.078,-177.325,10.914,149.502
C04540=1126.822,346.549,-82.043,-177.329,10.912,149.502
C04541=1126.826,346.301,-82.008,-177.332,10.910,149.502
C04542=1126.831,346.055,-81.973,-177.335,10.907,149.502
C04543=1126.835,345.806,-81.938,-177.338,10.904,149.502
C04544=1126.838,345.560,-81.903,-177.341,10.902,149.503
C04545=1126.842,345.312,-81.868,-177.345,10.899,149.503
C04546=1126.846,345.064,-81.834,-177.347,10.898,149.503
C04547=1126.850,344.817,-81.798,-177.351,10.895,149.503
C04548=1126.854,344.569,-81.764,-177.354,10.893,149.504
C04549=1126.858,344.322,-81.730,-177.357,10.890,149.504
C04550=1126.862,344.074,-81.694,-177.360,10.888,149.504
C04551=1126.866,343.827,-81.660,-177.364,10.885,149.504
C04552=1126.870,343.579,-81.626,-177.367,10.883,149.504
C04553=1126.873,343.331,-81.590,-177.370,10.880,149.505
C04554=1126.878,343.084,-81.556,-177.373,10.878,149.505
C04555=1126.882,342.836,-81.521,-177.376,10.875,149.505
C04556=1126.886,342.589,-81.487,-177.380,10.872,149.505
C04557=1126.889,342.341,-81.451,-177.383,10.870,149.505
C04558=1126.894,342.094,-81.417,-177.386,10.868,149.506
C04559=1126.897,341.846,-81.383,-177.390,10.865,149.506
C04560=1126.902,341.599,-81.348,-177.393,10.863,149.506
C04561=1126.906,341.351,-81.313,-177.396,10.860,149.506
C04562=1126.910,341.103,-81.279,-177.399,10.857,149.506
C04563=1126.913,340.856,-81.244,-177.403,10.855,149.507
C04564=1126.917,340.609,-81.210,-177.406,10.852,149.507
C04565=1126.921,340.361,-81.175,-177.409,10.850,149.507
C04566=1126.926,340.113,-81.141,-177.412,10.847,149.507
C04567=1126.929,339.865,-81.106,-177.415,10.845,149.507
C04568=1126.933,339.618,-81.072,-177.418,10.843,149.508
C04569=1126.937,339.370,-81.038,-177.421,10.841,149.508
C04570=1126.941,339.123,-81.003,-177.425,10.838,149.508
C04571=1126.944,338.875,-80.969,-177.428,10.835,149.508
C04572=1126.949,338.628,-80.935,-177.431,10.833,149.508
C04573=1126.954,338.380,-80.900,-177.434,10.831,149.509
C04574=1126.957,338.132,-80.866,-177.438,10.828,149.509
C04575=1126.961,337.885,-80.831,-177.441,10.826,149.509
C04576=1126.965,337.637,-80.797,-177.444,10.823,149.509
C04577=1126.969,337.390,-80.763,-177.447,10.820,149.509
C04578=1126.972,337.142,-80.728,-177.450,10.818,149.510
C04579=1126.976,336.895,-80.695,-177.454,10.815,149.510
C04580=1126.980,336.646,-80.660,-177.457,10.813,149.510
C04581=1126.984,336.399,-80.627,-177.460,10.810,149.510
C04582=1126.989,336.152,-80.592,-177.463,10.808,149.510
C04583=1126.992,335.904,-80.558,-177.467,10.805,149.511
C04584=1126.996,335.691,-80.529,-177.469,10.803,149.511
C04585=1127.000,335.478,-80.499,-177.472,10.801,149.511
C04586=1127.002,335.265,-80.470,-177.475,10.799,149.511
C04587=1127.006,335.052,-80.441,-177.477,10.797,149.511
C04588=1127.009,334.840,-80.411,-177.480,10.794,149.511
C04589=1127.013,334.627,-80.382,-177.483,10.793,149.512
C04590=1127.016,334.414,-80.353,-177.486,10.790,149.512
C04591=1127.020,334.201,-80.323,-177.488,10.788,149.512
C04592=1127.024,333.953,-80.290,-177.492,10.786,149.512
C04593=1127.028,333.706,-80.256,-177.495,10.783,149.512
C04594=1127.032,333.458,-80.221,-177.498,10.781,149.512
C04595=1127.035,333.210,-80.187,-177.501,10.778,149.513
C04596=1127.040,332.963,-80.154,-177.505,10.776,149.513
C04597=1127.043,332.715,-80.119,-177.508,10.773,149.513
C04598=1127.047,332.467,-80.085,-177.511,10.770,149.513
C04599=1127.051,332.220,-80.052,-177.514,10.768,149.513
C04600=1127.055,331.972,-80.018,-177.517,10.766,149.514
C04601=1127.060,331.724,-79.984,-177.520,10.764,149.514
C04602=1127.063,331.477,-79.950,-177.523,10.761,149.514
C04603=1127.067,331.229,-79.916,-177.526,10.759,149.514
C04604=1127.072,330.981,-79.882,-177.529,10.756,149.514
C04605=1127.075,330.734,-79.848,-177.533,10.753,149.515
C04606=1127.079,330.485,-79.815,-177.536,10.751,149.515
C04607=1127.083,330.238,-79.781,-177.539,10.749,149.515
C04608=1127.087,329.991,-79.748,-177.542,10.746,149.515
C04609=1127.091,329.743,-79.713,-177.546,10.743,149.515
C04610=1127.095,329.495,-79.680,-177.549,10.741,149.516
C04611=1127.099,329.248,-79.646,-177.552,10.738,149.516
C04612=1127.103,329.000,-79.613,-177.555,10.736,149.516
C04613=1127.107,328.752,-79.580,-177.558,10.733,149.516
C04614=1127.111,328.504,-79.545,-177.562,10.731,149.516
C04615=1127.115,328.256,-79.512,-177.565,10.728,149.516
C04616=1127.119,328.009,-79.478,-177.568,10.726,149.517
C04617=1127.123,327.761,-79.445,-177.571,10.723,149.517
C04618=1127.127,327.514,-79.411,-177.574,10.720,149.517
C04619=1127.130,327.266,-79.377,-177.577,10.719,149.517
C04620=1127.135,327.018,-79.344,-177.580,10.716,149.518
C04621=1127.140,326.770,-79.310,-177.583,10.713,149.518
C04622=1127.143,326.523,-79.276,-177.587,10.711,149.518
C04623=1127.147,326.275,-79.243,-177.590,10.709,149.518
C04624=1127.151,326.027,-79.210,-177.593,10.706,149.518
C04625=1127.155,325.779,-79.177,-177.596,10.703,149.518
C04626=1127.159,325.532,-79.143,-177.599,10.701,149.519
C04627=1127.163,325.284,-79.110,-177.603,10.698,149.519
C04628=1127.167,325.037,-79.076,-177.606,10.696,149.519
C04629=1127.171,324.788,-79.043,-177.609,10.693,149.519
C04630=1127.175,324.540,-79.010,-177.612,10.691,149.519
C04631=1127.179,324.293,-78.976,-177.615,10.688,149.519
C04632=1127.183,324.046,-78.943,-177.619,10.686,149.520
C04633=1127.187,323.798,-78.909,-177.622,10.683,149.520
C04634=1127.191,323.550,-78.876,-177.625,10.680,149.520
C04635=1127.195,323.302,-78.843,-177.628,10.678,149.520
C04636=1127.199,323.054,-78.810,-177.631,10.675,149.521
C04637=1127.203,322.806,-78.777,-177.634,10.673,149.521
C04638=1127.207,322.559,-78.743,-177.637,10.671,149.521
C04639=1127.211,322.311,-78.710,-177.640,10.669,149.521
C04640=1127.215,322.098,-78.681,-177.643,10.666,149.521
C04641=1127.218,321.885,-78.653,-177.646,10.664,149.521
C04642=1127.221,321.672,-78.625,-177.649,10.661,149.522
C04643=1127.225,321.459,-78.596,-177.651,10.659,149.522
C04644=1127.228,321.246,-78.567,-177.654,10.658,149.522
C04645=1127.232,321.033,-78.540,-177.657,10.655,149.522
C04646=1127.235,320.820,-78.511,-177.660,10.653,149.522
C04647=1127.239,320.607,-78.482,-177.662,10.651,149.522
C04648=1127.243,320.359,-78.449,-177.665,10.649,149.523
C04649=1127.247,320.112,-78.415,-177.668,10.646,149.523
C04650=1127.251,319.864,-78.384,-177.671,10.644,149.523
C04651=1127.255,319.616,-78.350,-177.675,10.641,149.523
C04652=1127.259,319.368,-78.317,-177.678,10.638,149.523
C04653=1127.263,319.120,-78.284,-177.681,10.636,149.524
C04654=1127.267,318.873,-78.251,-177.684,10.633,149.524
C04655=1127.271,318.625,-78.218,-177.687,10.631,149.524
C04656=1127.275,318.378,-78.185,-177.691,10.628,149.524
C04657=1127.279,318.128,-78.152,-177.694,10.625,149.524
C04658=1127.283,317.881,-78.119,-177.697,10.623,149.524
C04659=1127.287,317.633,-78.086,-177.700,10.621,149.525
C04660=1127.290,317.386,-78.054,-177.703,10.618,149.525
C04661=1127.294,317.138,-78.020,-177.706,10.615,149.525
C04662=1127.299,316.890,-77.988,-177.710,10.613,149.525
C04663=1127.303,316.642,-77.955,-177.713,10.610,149.525
C04664=1127.306,316.394,-77.922,-177.715,10.609,149.526
C04665=1127.311,316.147,-77.890,-177.718,10.606,149.526
C04666=1127.315,315.899,-77.857,-177.722,10.603,149.526
C04667=1127.319,315.652,-77.824,-177.725,10.601,149.526
C04668=1127.323,315.403,-77.792,-177.728,10.598,149.526
C04669=1127.327,315.156,-77.759,-177.731,10.596,149.526
C04670=1127.331,314.908,-77.726,-177.734,10.593,149.527
C04671=1127.335,314.660,-77.694,-177.737,10.590,149.527
C04672=1127.339,314.412,-77.661,-177.741,10.588,149.527
C04673=1127.343,314.165,-77.628,-177.744,10.585,149.527
C04674=1127.347,313.916,-77.596,-177.747,10.583,149.527
C04675=1127.351,313.669,-77.563,-177.750,10.580,149.527
C04676=1127.355,313.420,-77.531,-177.753,10.578,149.528
C04677=1127.359,313.173,-77.498,-177.757,10.575,149.528
C04678=1127.364,312.924,-77.465,-177.760,10.572,149.528
C04679=1127.367,312.677,-77.433,-177.763,10.570,149.528
C04680=1127.372,312.429,-77.400,-177.765,10.568,149.528
C04681=1127.376,312.182,-77.368,-177.769,10.565,149.529
C04682=1127.380,311.934,-77.335,-177.772,10.563,149.529
C04683=1127.383,311.686,-77.303,-177.775,10.560,149.529
C04684=1127.388,311.438,-77.270,-177.778,10.558,149.529
C04685=1127.392,311.189,-77.238,-177.781,10.555,149.529
C04686=1127.396,310.942,-77.205,-177.784,10.553,149.530
C04687=1127.400,310.694,-77.173,-177.788,10.550,149.530
C04688=1127.404,310.447,-77.141,-177.791,10.547,149.530
C04689=1127.409,310.199,-77.108,-177.794,10.545,149.530
C04690=1127.412,309.951,-77.077,-177.797,10.542,149.530
C04691=1127.416,309.703,-77.043,-177.800,10.540,149.531
C04692=1127.420,309.455,-77.012,-177.803,10.537,149.531
C04693=1127.425,309.206,-76.979,-177.806,10.535,149.531
C04694=1127.429,308.960,-76.947,-177.810,10.532,149.531
C04695=1127.433,308.711,-76.914,-177.812,10.530,149.531
C04696=1127.436,308.498,-76.887,-177.815,10.527,149.531
C04697=1127.439,308.285,-76.859,-177.818,10.526,149.532
C04698=1127.443,308.071,-76.831,-177.821,10.523,149.532
C04699=1127.447,307.859,-76.804,-177.823,10.521,149.532
C04700=1127.451,307.645,-76.776,-177.826,10.519,149.532
C04701=1127.454,307.432,-76.748,-177.829,10.517,149.532
C04702=1127.457,307.218,-76.721,-177.831,10.515,149.532
C04703=1127.461,307.006,-76.694,-177.834,10.513,149.533
C04704=1127.465,306.758,-76.661,-177.837,10.510,149.533
C04705=1127.469,306.510,-76.629,-177.840,10.508,149.533
C04706=1127.473,306.262,-76.597,-177.843,10.505,149.533
C04707=1127.477,306.015,-76.565,-177.846,10.502,149.533
C04708=1127.482,305.766,-76.533,-177.849,10.500,149.533
C04709=1127.485,305.518,-76.501,-177.852,10.497,149.534
C04710=1127.489,305.270,-76.469,-177.856,10.495,149.534
C04711=1127.494,305.022,-76.437,-177.859,10.492,149.534
C04712=1127.498,304.774,-76.405,-177.862,10.490,149.534
C04713=1127.502,304.526,-76.373,-177.865,10.487,149.534
C04714=1127.507,304.279,-76.341,-177.868,10.484,149.535
C04715=1127.510,304.031,-76.309,-177.871,10.482,149.535
C04716=1127.514,303.783,-76.278,-177.875,10.479,149.535
C04717=1127.518,303.535,-76.246,-177.877,10.477,149.535
C04718=1127.523,303.287,-76.214,-177.880,10.475,149.535
C04719=1127.527,303.039,-76.182,-177.883,10.472,149.535
C04720=1127.530,302.791,-76.150,-177.886,10.470,149.536
C04721=1127.535,302.543,-76.118,-177.890,10.467,149.536
C04722=1127.539,302.295,-76.086,-177.893,10.464,149.536
C04723=1127.543,302.048,-76.055,-177.896,10.462,149.536
C04724=1127.547,301.800,-76.023,-177.899,10.459,149.536
C04725=1127.551,301.552,-75.991,-177.902,10.457,149.537
C04726=1127.556,301.304,-75.960,-177.905,10.454,149.537
C04727=1127.560,301.055,-75.928,-177.909,10.452,149.537
C04728=1127.563,300.807,-75.896,-177.911,10.449,149.537
C04729=1127.568,300.560,-75.864,-177.915,10.446,149.537
C04730=1127.572,300.312,-75.832,-177.917,10.444,149.537
C04731=1127.576,300.064,-75.800,-177.920,10.442,149.538
C04732=1127.581,299.816,-75.769,-177.923,10.439,149.538
C04733=1127.584,299.568,-75.737,-177.927,10.437,149.538
C04734=1127.589,299.320,-75.706,-177.930,10.434,149.538
C04735=1127.592,299.072,-75.674,-177.933,10.432,149.538
C04736=1127.596,298.824,-75.643,-177.936,10.429,149.538
C04737=1127.601,298.576,-75.612,-177.939,10.426,149.539
C04738=1127.604,298.328,-75.580,-177.942,10.424,149.539
C04739=1127.609,298.080,-75.549,-177.946,10.421,149.539
C04740=1127.613,297.832,-75.516,-177.948,10.418,149.539
C04741=1127.618,297.585,-75.485,-177.952,10.416,149.539
C04742=1127.622,297.336,-75.454,-177.955,10.413,149.539
C04743=1127.625,297.088,-75.422,-177.957,10.412,149.540
C04744=1127.630,296.840,-75.391,-177.960,10.409,149.540
C04745=1127.634,296.592,-75.359,-177.964,10.406,149.540
C04746=1127.638,296.345,-75.328,-177.967,10.404,149.540
C04747=1127.642,296.096,-75.297,-177.970,10.401,149.540
C04748=1127.646,295.849,-75.265,-177.973,10.398,149.541
C04749=1127.650,295.600,-75.234,-177.976,10.396,149.541
C04750=1127.655,295.353,-75.203,-177.979,10.393,149.541
C04751=1127.659,295.104,-75.172,-177.982,10.391,149.541
C04752=1127.662,294.892,-75.144,-177.985,10.389,149.541
C04753=1127.666,294.678,-75.117,-177.988,10.386,149.541
C04754=1127.669,294.464,-75.091,-177.990,10.384,149.542
C04755=1127.673,294.251,-75.064,-177.993,10.382,149.542
C04756=1127.676,294.038,-75.037,-177.996,10.380,149.542
C04757=1127.680,293.824,-75.010,-177.998,10.378,149.542
C04758=1127.684,293.611,-74.983,-178.001,10.376,149.542
C04759=1127.687,293.398,-74.957,-178.004,10.373,149.542
C04760=1127.691,293.150,-74.925,-178.007,10.371,149.542
C04761=1127.695,292.902,-74.895,-178.010,10.368,149.543
C04762=1127.699,292.653,-74.864,-178.012,10.366,149.543
C04763=1127.704,292.406,-74.832,-178.016,10.364,149.543
C04764=1127.708,292.157,-74.801,-178.018,10.361,149.543
C04765=1127.712,291.909,-74.770,-178.022,10.359,149.543
C04766=1127.716,291.661,-74.738,-178.025,10.356,149.544
C04767=1127.720,291.414,-74.708,-178.028,10.353,149.544
C04768=1127.724,291.166,-74.677,-178.031,10.351,149.544
C04769=1127.728,290.918,-74.646,-178.034,10.348,149.544
C04770=1127.733,290.670,-74.615,-178.037,10.345,149.544
C04771=1127.737,290.421,-74.584,-178.041,10.343,149.545
C04772=1127.741,290.173,-74.554,-178.044,10.340,149.545
C04773=1127.744,289.925,-74.522,-178.046,10.338,149.545
C04774=1127.749,289.677,-74.491,-178.049,10.336,149.545
C04775=1127.753,289.429,-74.460,-178.052,10.333,149.545
C04776=1127.758,289.181,-74.429,-178.055,10.331,149.545
C04777=1127.761,288.933,-74.399,-178.058,10.328,149.545
C04778=1127.765,288.684,-74.368,-178.062,10.325,149.546
C04779=1127.770,288.437,-74.336,-178.065,10.323,149.546
C04780=1127.774,288.189,-74.306,-178.068,10.320,149.546
C04781=1127.778,287.941,-74.275,-178.071,10.317,149.546
C04782=1127.782,287.693,-74.244,-178.074,10.315,149.547
C04783=1127.787,287.445,-74.213,-178.077,10.312,149.547
C04784=1127.790,287.196,-74.183,-178.080,10.310,149.547
C04785=1127.795,286.948,-74.152,-178.083,10.308,149.547
C04786=1127.799,286.701,-74.121,-178.086,10.305,149.547
C04787=1127.803,286.452,-74.091,-178.089,10.303,149.547
C04788=1127.807,286.204,-74.060,-178.092,10.300,149.547
C04789=1127.812,285.956,-74.029,-178.095,10.298,149.548
C04790=1127.815,285.708,-73.999,-178.098,10.295,149.548
C04791=1127.820,285.460,-73.968,-178.102,10.292,149.548
C04792=1127.824,285.212,-73.937,-178.105,10.290,149.548
C04793=1127.828,284.964,-73.907,-178.108,10.287,149.548
C04794=1127.832,284.716,-73.876,-178.110,10.285,149.549
C04795=1127.836,284.468,-73.846,-178.113,10.282,149.549
C04796=1127.841,284.220,-73.815,-178.117,10.280,149.549
C04797=1127.845,283.971,-73.785,-178.120,10.277,149.549
C04798=1127.849,283.723,-73.754,-178.123,10.275,149.549
C04799=1127.853,283.475,-73.724,-178.126,10.272,149.549
C04800=1127.857,283.228,-73.693,-178.129,10.269,149.550
C04801=1127.861,282.979,-73.662,-178.132,10.267,149.550
C04802=1127.865,282.731,-73.632,-178.135,10.264,149.550
C04803=1127.870,282.483,-73.602,-178.138,10.262,149.550
C04804=1127.874,282.235,-73.572,-178.141,10.260,149.550
C04805=1127.879,281.987,-73.541,-178.144,10.257,149.551
C04806=1127.882,281.739,-73.511,-178.147,10.255,149.551
C04807=1127.887,281.490,-73.481,-178.150,10.252,149.551
C04808=1127.891,281.277,-73.454,-178.153,10.249,149.551
C04809=1127.894,281.064,-73.428,-178.156,10.247,149.551
C04810=1127.898,280.850,-73.402,-178.160,10.244,149.551
C04811=1127.901,280.637,-73.376,-178.162,10.242,149.552
C04812=1127.905,280.423,-73.350,-178.165,10.240,149.552
C04813=1127.908,280.210,-73.324,-178.168,10.237,149.552
C04814=1127.912,279.996,-73.298,-178.171,10.235,149.552
C04815=1127.916,279.782,-73.272,-178.174,10.233,149.552
C04816=1127.920,279.535,-73.241,-178.178,10.229,149.553
C04817=1127.924,279.286,-73.212,-178.181,10.227,149.553
C04818=1127.928,279.038,-73.181,-178.185,10.223,149.553
C04819=1127.933,278.790,-73.152,-178.188,10.221,149.553
C04820=1127.937,278.542,-73.121,-178.191,10.218,149.553
C04821=1127.941,278.293,-73.091,-178.194,10.216,149.554
C04822=1127.945,278.045,-73.061,-178.198,10.212,149.554
C04823=1127.950,277.797,-73.031,-178.201,10.210,149.554
C04824=1127.953,277.549,-73.001,-178.204,10.207,149.554
C04825=1127.958,277.301,-72.971,-178.207,10.204,149.554
C04826=1127.962,277.053,-72.940,-178.211,10.201,149.554
C04827=1127.966,276.805,-72.911,-178.214,10.198,149.555
C04828=1127.970,276.557,-72.881,-178.217,10.196,149.555
C04829=1127.974,276.308,-72.851,-178.220,10.193,149.555
C04830=1127.979,276.060,-72.820,-178.223,10.191,149.555
C04831=1127.983,275.812,-72.791,-178.227,10.188,149.555
C04832=1127.987,275.564,-72.761,-178.230,10.185,149.555
C04833=1127.991,275.316,-72.731,-178.233,10.182,149.556
C04834=1127.996,275.067,-72.701,-178.236,10.179,149.556
C04835=1128.000,274.819,-72.672,-178.239,10.177,149.556
C04836=1128.004,274.572,-72.642,-178.242,10.174,149.556
C04837=1128.008,274.323,-72.612,-178.245,10.171,149.556
C04838=1128.013,274.075,-72.582,-178.248,10.168,149.556
C04839=1128.017,273.827,-72.552,-178.252,10.166,149.557
C04840=1128.021,273.579,-72.522,-178.254,10.163,149.557
C04841=1128.025,273.331,-72.493,-178.257,10.160,149.557
C04842=1128.029,273.082,-72.464,-178.260,10.158,149.557
C04843=1128.033,272.835,-72.433,-178.263,10.155,149.557
C04844=1128.038,272.586,-72.403,-178.266,10.152,149.557
C04845=1128.042,272.338,-72.374,-178.269,10.149,149.557
C04846=1128.046,272.089,-72.344,-178.271,10.147,149.557
C04847=1128.051,271.841,-72.315,-178.275,10.145,149.558
C04848=1128.055,271.593,-72.285,-178.278,10.142,149.558
C04849=1128.059,271.345,-72.255,-178.281,10.140,149.558
C04850=1128.063,271.097,-72.226,-178.284,10.137,149.558
C04851=1128.067,270.849,-72.196,-178.287,10.134,149.558
C04852=1128.071,270.600,-72.167,-178.289,10.132,149.558
C04853=1128.076,270.352,-72.137,-178.292,10.129,149.558
C04854=1128.080,270.104,-72.107,-178.295,10.127,149.558
C04855=1128.084,269.855,-72.078,-178.298,10.124,149.558
C04856=1128.089,269.607,-72.049,-178.300,10.122,149.559
C04857=1128.093,269.359,-72.019,-178.303,10.119,149.559
C04858=1128.097,269.111,-71.990,-178.306,10.116,149.559
C04859=1128.101,268.862,-71.960,-178.308,10.114,149.559
C04860=1128.105,268.614,-71.931,-178.311,10.111,149.559
C04861=1128.110,268.366,-71.901,-178.314,10.108,149.559
C04862=1128.114,268.117,-71.872,-178.316,10.106,149.559
C04863=1128.119,267.870,-71.843,-178.319,10.104,149.559
C04864=1128.121,267.656,-71.817,-178.321,10.102,149.559
C04865=1128.125,267.442,-71.792,-178.324,10.100,149.559
C04866=1128.129,267.229,-71.767,-178.326,10.098,149.559
C04867=1128.133,267.015,-71.741,-178.328,10.095,149.559
C04868=1128.136,266.802,-71.716,-178.330,10.093,149.560
C04869=1128.140,266.588,-71.691,-178.332,10.091,149.560
C04870=1128.144,266.374,-71.666,-178.335,10.089,149.560
C04871=1128.147,266.161,-71.641,-178.337,10.087,149.560
C04872=1128.152,265.913,-71.612,-178.339,10.084,149.560
C04873=1128.156,265.664,-71.582,-178.342,10.082,149.560
C04874=1128.160,265.416,-71.553,-178.344,10.080,149.560
C04875=1128.164,265.168,-71.523,-178.347,10.078,149.560
C04876=1128.169,264.919,-71.494,-178.349,10.076,149.560
C04877=1128.173,264.671,-71.465,-178.352,10.074,149.560
C04878=1128.178,264.423,-71.436,-178.355,10.071,149.561
C04879=1128.182,264.175,-71.406,-178.358,10.067,149.561
C04880=1128.186,263.926,-71.378,-178.362,10.064,149.561
C04881=1128.190,263.678,-71.349,-178.366,10.061,149.561
C04882=1128.194,263.430,-71.319,-178.369,10.059,149.561
C04883=1128.199,263.182,-71.290,-178.373,10.055,149.562
C04884=1128.203,262.933,-71.262,-178.377,10.052,149.562
C04885=1128.207,262.685,-71.232,-178.381,10.049,149.562
C04886=1128.211,262.437,-71.203,-178.384,10.046,149.562
C04887=1128.215,262.188,-71.175,-178.388,10.043,149.563
C04888=1128.220,261.941,-71.145,-178.392,10.039,149.563
C04889=1128.224,261.692,-71.116,-178.395,10.037,149.563
C04890=1128.229,261.443,-71.087,-178.398,10.033,149.563
C04891=1128.232,261.196,-71.058,-178.402,10.031,149.563
C04892=1128.237,260.947,-71.030,-178.405,10.027,149.563
C04893=1128.242,260.699,-71.001,-178.409,10.024,149.563
C04894=1128.246,260.450,-70.972,-178.412,10.021,149.564
C04895=1128.249,260.202,-70.943,-178.416,10.018,149.564
C04896=1128.255,259.954,-70.915,-178.419,10.015,149.564
C04897=1128.259,259.706,-70.885,-178.422,10.012,149.564
C04898=1128.262,259.457,-70.857,-178.426,10.009,149.564
C04899=1128.267,259.210,-70.828,-178.429,10.007,149.564
C04900=1128.272,258.961,-70.799,-178.432,10.004,149.565
C04901=1128.275,258.713,-70.770,-178.435,10.000,149.565
C04902=1128.280,258.464,-70.742,-178.438,9.997,149.565
C04903=1128.285,258.216,-70.713,-178.441,9.995,149.565
C04904=1128.288,257.968,-70.684,-178.444,9.992,149.565
C04905=1128.293,257.719,-70.656,-178.448,9.988,149.565
C04906=1128.297,257.471,-70.628,-178.451,9.986,149.565
C04907=1128.301,257.223,-70.598,-178.454,9.983,149.565
C04908=1128.306,256.974,-70.570,-178.456,9.980,149.565
C04909=1128.310,256.726,-70.542,-178.459,9.977,149.566
C04910=1128.314,256.478,-70.512,-178.462,9.974,149.565
C04911=1128.318,256.229,-70.484,-178.465,9.972,149.566
C04912=1128.323,255.981,-70.456,-178.468,9.969,149.566
C04913=1128.327,255.732,-70.428,-178.468,9.967,149.565
C04914=1128.332,255.485,-70.399,-178.467,9.967,149.565
C04915=1128.335,255.236,-70.371,-178.467,9.965,149.565
C04916=1128.340,254.987,-70.342,-178.467,9.965,149.564
C04917=1128.345,254.739,-70.313,-178.467,9.964,149.564
C04918=1128.348,254.491,-70.285,-178.467,9.963,149.564
C04919=1128.353,254.242,-70.256,-178.468,9.961,149.564
C04920=1128.356,254.029,-70.232,-178.469,9.960,149.564
C04921=1128.360,253.816,-70.207,-178.470,9.959,149.564
C04922=1128.364,253.602,-70.183,-178.471,9.957,149.564
C04923=1128.368,253.388,-70.158,-178.473,9.956,149.564
C04924=1128.372,253.174,-70.134,-178.474,9.955,149.564
C04925=1128.375,252.961,-70.109,-178.476,9.952,149.564
C04926=1128.378,252.747,-70.085,-178.478,9.951,149.564
C04927=1128.382,252.532,-70.060,-178.480,9.949,149.564
C04928=1128.387,252.285,-70.032,-178.483,9.947,149.564
C04929=1128.391,252.036,-70.004,-178.486,9.944,149.564
C04930=1128.395,251.788,-69.975,-178.489,9.942,149.565
C04931=1128.400,251.540,-69.947,-178.492,9.938,149.565
C04932=1128.403,251.291,-69.918,-178.496,9.936,149.565
C04933=1128.409,251.043,-69.890,-178.500,9.933,149.565
C04934=1128.412,250.794,-69.862,-178.504,9.930,149.566
C04935=1128.417,250.545,-69.833,-178.508,9.927,149.566
C04936=1128.421,250.297,-69.805,-178.513,9.923,149.567
C04937=1128.425,250.049,-69.777,-178.517,9.919,149.567
C04938=1128.430,249.801,-69.749,-178.522,9.915,149.567
C04939=1128.434,249.552,-69.721,-178.528,9.912,149.568
C04940=1128.439,249.304,-69.692,-178.533,9.907,149.568
C04941=1128.443,249.055,-69.664,-178.538,9.903,149.568
C04942=1128.447,248.808,-69.636,-178.545,9.899,149.569
C04943=1128.451,248.559,-69.608,-178.551,9.894,149.570
C04944=1128.456,248.311,-69.580,-178.557,9.888,149.570
C04945=1128.460,248.062,-69.552,-178.564,9.884,149.571
C04946=1128.464,247.814,-69.525,-178.570,9.879,149.571
C04947=1128.469,247.565,-69.496,-178.578,9.873,149.572
C04948=1128.473,247.317,-69.468,-178.582,9.869,149.572
C04949=1128.477,247.069,-69.440,-178.584,9.866,149.572
C04950=1128.481,246.820,-69.413,-178.585,9.864,149.571
C04951=1128.486,246.572,-69.385,-178.585,9.863,149.571
C04952=1128.490,246.323,-69.356,-178.587,9.860,149.571
C04953=1128.495,246.075,-69.329,-178.588,9.858,149.571
C04954=1128.499,245.827,-69.302,-178.590,9.856,149.571
C04955=1128.503,245.578,-69.273,-178.591,9.853,149.571
C04956=1128.508,245.330,-69.246,-178.593,9.852,149.571
C04957=1128.511,245.081,-69.218,-178.595,9.849,149.570
C04958=1128.516,244.833,-69.190,-178.595,9.847,149.570
C04959=1128.521,244.584,-69.163,-178.597,9.845,149.570
C04960=1128.525,244.336,-69.135,-178.599,9.843,149.570
C04961=1128.529,244.088,-69.107,-178.601,9.840,149.570
C04962=1128.533,243.839,-69.079,-178.602,9.839,149.570
C04963=1128.538,243.591,-69.052,-178.604,9.837,149.570
C04964=1128.542,243.343,-69.024,-178.606,9.834,149.570
C04965=1128.547,243.093,-68.996,-178.608,9.832,149.570
C04966=1128.551,242.846,-68.968,-178.610,9.830,149.570
C04967=1128.556,242.597,-68.941,-178.612,9.827,149.570
C04968=1128.560,242.349,-68.913,-178.614,9.825,149.570
C04969=1128.564,242.100,-68.886,-178.616,9.823,149.570
C04970=1128.569,241.852,-68.858,-178.618,9.821,149.570
C04971=1128.573,241.603,-68.831,-178.620,9.818,149.570
C04972=1128.577,241.355,-68.803,-178.622,9.816,149.570
C04973=1128.582,241.107,-68.776,-178.624,9.814,149.570
C04974=1128.585,240.858,-68.748,-178.626,9.812,149.570
C04975=1128.590,240.610,-68.721,-178.629,9.808,149.570
C04976=1128.594,240.395,-68.696,-178.631,9.807,149.570
C04977=1128.598,240.182,-68.673,-178.632,9.805,149.570
C04978=1128.602,239.968,-68.649,-178.634,9.803,149.570
C04979=1128.605,239.754,-68.625,-178.636,9.801,149.570
C04980=1128.609,239.540,-68.602,-178.638,9.798,149.570
C04981=1128.613,239.326,-68.578,-178.641,9.796,149.570
C04982=1128.616,239.113,-68.554,-178.642,9.794,149.570
C04983=1128.620,238.899,-68.531,-178.645,9.792,149.570
C04984=1128.624,238.650,-68.503,-178.647,9.790,149.570
C04985=1128.628,238.402,-68.476,-178.650,9.787,149.570
C04986=1128.633,238.153,-68.449,-178.653,9.784,149.570
C04987=1128.637,237.905,-68.421,-178.655,9.782,149.570
C04988=1128.642,237.656,-68.394,-178.657,9.779,149.570
C04989=1128.646,237.408,-68.367,-178.660,9.776,149.570
C04990=1128.651,237.160,-68.339,-178.663,9.774,149.571
C04991=1128.655,236.911,-68.311,-178.666,9.772,149.571
C04992=1128.659,236.662,-68.284,-178.669,9.769,149.571
C04993=1128.664,236.414,-68.257,-178.671,9.766,149.571
C04994=1128.668,236.166,-68.229,-178.674,9.763,149.571
C04995=1128.672,235.917,-68.202,-178.677,9.760,149.571
C04996=1128.677,235.668,-68.175,-178.680,9.758,149.571
C04997=1128.681,235.420,-68.147,-178.683,9.755,149.571
C04998=1128.685,235.172,-68.121,-178.686,9.752,149.571
C04999=1128.690,234.924,-68.094,-178.689,9.749,149.571
C05000=1128.694,234.674,-68.066,-178.692,9.747,149.572
C05001=1128.699,234.426,-68.039,-178.695,9.744,149.572
C05002=1128.703,234.178,-68.011,-178.698,9.741,149.572
C05003=1128.708,233.930,-67.984,-178.701,9.739,149.572
C05004=1128.712,233.681,-67.958,-178.705,9.735,149.572
C05005=1128.716,233.432,-67.930,-178.707,9.732,149.572
C05006=1128.720,233.184,-67.903,-178.710,9.730,149.573
C05007=1128.725,232.935,-67.876,-178.714,9.726,149.573
C05008=1128.730,232.687,-67.849,-178.717,9.723,149.573
C05009=1128.733,232.439,-67.823,-178.721,9.720,149.573
C05010=1128.738,232.190,-67.796,-178.723,9.717,149.573
C05011=1128.742,231.941,-67.768,-178.727,9.714,149.573
C05012=1128.747,231.692,-67.741,-178.731,9.710,149.573
C05013=1128.751,231.444,-67.715,-178.734,9.708,149.574
C05014=1128.755,231.196,-67.688,-178.738,9.704,149.574
C05015=1128.760,230.947,-67.661,-178.741,9.701,149.574
C05016=1128.764,230.699,-67.634,-178.745,9.697,149.574
C05017=1128.769,230.450,-67.607,-178.748,9.695,149.574
C05018=1128.773,230.202,-67.580,-178.752,9.691,149.574
C05019=1128.778,229.953,-67.553,-178.756,9.687,149.574
C05020=1128.781,229.705,-67.526,-178.760,9.684,149.575
C05021=1128.786,229.456,-67.499,-178.763,9.680,149.575
C05022=1128.790,229.207,-67.473,-178.767,9.677,149.575
C05023=1128.795,228.959,-67.446,-178.771,9.673,149.575
C05024=1128.799,228.710,-67.419,-178.774,9.670,149.575
C05025=1128.803,228.462,-67.393,-178.777,9.667,149.575
C05026=1128.808,228.214,-67.366,-178.781,9.663,149.575
C05027=1128.812,227.965,-67.340,-178.784,9.660,149.576
C05028=1128.817,227.716,-67.313,-178.788,9.656,149.576
C05029=1128.822,227.468,-67.286,-178.792,9.653,149.576
C05030=1128.825,227.220,-67.259,-178.795,9.649,149.576
C05031=1128.830,226.971,-67.233,-178.799,9.646,149.576
C05032=1128.834,226.757,-67.210,-178.801,9.643,149.576
C05033=1128.838,226.543,-67.187,-178.804,9.640,149.576
C05034=1128.841,226.329,-67.165,-178.807,9.637,149.576
C05035=1128.845,226.115,-67.142,-178.810,9.634,149.576
C05036=1128.849,225.901,-67.119,-178.813,9.631,149.576
C05037=1128.853,225.688,-67.096,-178.815,9.628,149.576
C05038=1128.857,225.473,-67.074,-178.818,9.626,149.576
C05039=1128.861,225.259,-67.051,-178.821,9.622,149.576
C05040=1128.865,225.010,-67.024,-178.824,9.620,149.576
C05041=1128.869,224.762,-66.998,-178.827,9.616,149.576
C05042=1128.873,224.513,-66.972,-178.829,9.613,149.576
C05043=1128.878,224.264,-66.945,-178.833,9.609,149.576
C05044=1128.882,224.016,-66.919,-178.835,9.606,149.576
C05045=1128.887,223.767,-66.892,-178.839,9.603,149.577
C05046=1128.891,223.519,-66.866,-178.841,9.599,149.576
C05047=1128.895,223.270,-66.840,-178.845,9.596,149.576
C05048=1128.900,223.021,-66.813,-178.847,9.592,149.576
C05049=1128.905,222.773,-66.788,-178.850,9.590,149.576
C05050=1128.909,222.525,-66.761,-178.853,9.586,149.576
C05051=1128.914,222.276,-66.735,-178.856,9.583,149.576
C05052=1128.918,222.027,-66.709,-178.858,9.580,149.576
C05053=1128.923,221.779,-66.682,-178.861,9.577,149.576
C05054=1128.927,221.530,-66.656,-178.864,9.573,149.576
C05055=1128.931,221.281,-66.631,-178.867,9.570,149.576
C05056=1128.936,221.033,-66.604,-178.869,9.566,149.576
C05057=1128.941,220.785,-66.578,-178.872,9.563,149.576
C05058=1128.945,220.536,-66.552,-178.874,9.560,149.576
C05059=1128.949,220.288,-66.526,-178.877,9.557,149.576
C05060=1128.954,220.038,-66.500,-178.879,9.554,149.576
C05061=1128.958,219.790,-66.474,-178.882,9.551,149.576
C05062=1128.962,219.541,-66.448,-178.884,9.548,149.576
C05063=1128.967,219.293,-66.422,-178.887,9.545,149.576
C05064=1128.972,219.044,-66.396,-178.889,9.542,149.575
C05065=1128.976,218.795,-66.370,-178.892,9.538,149.575
C05066=1128.980,218.547,-66.344,-178.894,9.535,149.575
C05067=1128.984,218.298,-66.318,-178.896,9.533,149.575
C05068=1128.989,218.050,-66.292,-178.898,9.530,149.575
C05069=1128.994,217.801,-66.266,-178.901,9.526,149.575
C05070=1128.998,217.552,-66.240,-178.903,9.523,149.575
C05071=1129.002,217.304,-66.215,-178.905,9.521,149.575
C05072=1129.006,217.055,-66.189,-178.907,9.518,149.575
C05073=1129.011,216.807,-66.163,-178.909,9.515,149.574
C05074=1129.015,216.559,-66.137,-178.911,9.512,149.574
C05075=1129.020,216.309,-66.111,-178.914,9.509,149.574
C05076=1129.024,216.061,-66.085,-178.915,9.506,149.574
C05077=1129.029,215.813,-66.059,-178.918,9.503,149.574
C05078=1129.033,215.564,-66.034,-178.919,9.500,149.574
C05079=1129.038,215.315,-66.008,-178.921,9.498,149.574
C05080=1129.042,215.066,-65.982,-178.923,9.494,149.573
C05081=1129.047,214.818,-65.957,-178.925,9.492,149.573
C05082=1129.051,214.569,-65.931,-178.927,9.490,149.573
C05083=1129.055,214.320,-65.905,-178.929,9.486,149.573
C05084=1129.059,214.072,-65.880,-178.931,9.484,149.573
C05085=1129.065,213.823,-65.854,-178.933,9.481,149.573
C05086=1129.069,213.574,-65.828,-178.935,9.479,149.573
C05087=1129.073,213.326,-65.802,-178.936,9.476,149.572
C05088=1129.077,213.112,-65.781,-178.937,9.473,149.572
C05089=1129.081,212.897,-65.759,-178.939,9.471,149.572
C05090=1129.085,212.684,-65.736,-178.940,9.469,149.572
C05091=1129.088,212.469,-65.714,-178.942,9.467,149.572
C05092=1129.093,212.255,-65.692,-178.943,9.465,149.572
C05093=1129.096,212.041,-65.670,-178.945,9.463,149.572
C05094=1129.100,211.827,-65.648,-178.947,9.460,149.572
C05095=1129.104,211.613,-65.626,-178.948,9.459,149.572
C05096=1129.108,211.364,-65.600,-178.949,9.456,149.571
C05097=1129.112,211.116,-65.575,-178.952,9.453,149.571
C05098=1129.117,210.867,-65.549,-178.954,9.451,149.571
C05099=1129.122,210.618,-65.524,-178.956,9.448,149.571
C05100=1129.126,210.369,-65.498,-178.958,9.446,149.571
C05101=1129.131,210.121,-65.473,-178.960,9.443,149.571
C05102=1129.135,209.872,-65.447,-178.962,9.440,149.571
C05103=1129.139,209.624,-65.422,-178.964,9.438,149.571
C05104=1129.144,209.375,-65.396,-178.967,9.435,149.571
C05105=1129.149,209.126,-65.371,-178.968,9.433,149.571
C05106=1129.153,208.878,-65.346,-178.971,9.430,149.571
C05107=1129.158,208.629,-65.320,-178.973,9.428,149.571
C05108=1129.162,208.380,-65.294,-178.976,9.424,149.571
C05109=1129.167,208.132,-65.270,-178.978,9.422,149.571
C05110=1129.171,207.883,-65.244,-178.981,9.419,149.571
C05111=1129.175,207.634,-65.218,-178.983,9.416,149.571
C05112=1129.180,207.386,-65.193,-178.985,9.414,149.571
C05113=1129.184,207.137,-65.168,-178.988,9.411,149.571
C05114=1129.189,206.889,-65.143,-178.991,9.408,149.571
C05115=1129.193,206.640,-65.117,-178.993,9.406,149.571
C05116=1129.198,206.391,-65.092,-178.996,9.403,149.571
C05117=1129.202,206.142,-65.067,-178.998,9.400,149.571
C05118=1129.207,205.893,-65.041,-179.001,9.398,149.571
C05119=1129.212,205.645,-65.016,-179.004,9.394,149.571
C05120=1129.215,205.396,-64.991,-179.007,9.392,149.572
C05121=1129.220,205.148,-64.966,-179.010,9.389,149.572
C05122=1129.225,204.899,-64.941,-179.013,9.386,149.572
C05123=1129.230,204.651,-64.915,-179.015,9.383,149.572
C05124=1129.234,204.401,-64.890,-179.018,9.380,149.572
C05125=1129.238,204.153,-64.865,-179.021,9.378,149.572
C05126=1129.243,203.904,-64.840,-179.025,9.374,149.572
C05127=1129.247,203.656,-64.815,-179.028,9.371,149.572
C05128=1129.252,203.406,-64.790,-179.031,9.369,149.572
C05129=1129.256,203.159,-64.765,-179.034,9.365,149.572
C05130=1129.261,202.909,-64.740,-179.037,9.362,149.573
C05131=1129.265,202.660,-64.714,-179.040,9.359,149.573
C05132=1129.270,202.412,-64.690,-179.043,9.356,149.573
C05133=1129.274,202.163,-64.666,-179.046,9.353,149.573
C05134=1129.279,201.915,-64.640,-179.050,9.350,149.573
C05135=1129.284,201.666,-64.615,-179.053,9.347,149.573
C05136=1129.287,201.417,-64.590,-179.056,9.343,149.573
C05137=1129.292,201.169,-64.565,-179.060,9.340,149.574
C05138=1129.297,200.919,-64.540,-179.063,9.337,149.574
C05139=1129.301,200.671,-64.516,-179.066,9.333,149.574
C05140=1129.306,200.422,-64.491,-179.070,9.330,149.574
C05141=1129.310,200.174,-64.466,-179.074,9.326,149.574
C05142=1129.314,199.925,-64.441,-179.077,9.323,149.574
C05143=1129.319,199.676,-64.416,-179.081,9.319,149.574
C05144=1129.323,199.461,-64.395,-179.084,9.317,149.575
C05145=1129.327,199.247,-64.374,-179.087,9.314,149.575
C05146=1129.330,199.033,-64.352,-179.090,9.310,149.575
C05147=1129.334,198.819,-64.332,-179.093,9.308,149.575
C05148=1129.338,198.605,-64.310,-179.097,9.304,149.575
C05149=1129.343,198.390,-64.289,-179.100,9.301,149.575
C05150=1129.346,198.176,-64.267,-179.103,9.298,149.575
C05151=1129.350,197.961,-64.246,-179.106,9.295,149.576
C05152=1129.354,197.714,-64.222,-179.110,9.292,149.576
C05153=1129.359,197.465,-64.197,-179.114,9.287,149.576
C05154=1129.363,197.216,-64.173,-179.118,9.284,149.576
C05155=1129.368,196.967,-64.148,-179.122,9.280,149.576
C05156=1129.373,196.719,-64.124,-179.125,9.276,149.576
C05157=1129.377,196.469,-64.099,-179.130,9.272,149.576
C05158=1129.382,196.221,-64.075,-179.133,9.268,149.577
C05159=1129.387,195.972,-64.050,-179.135,9.266,149.576
C05160=1129.390,195.723,-64.026,-179.136,9.264,149.576
C05161=1129.395,195.475,-64.002,-179.137,9.261,149.576
C05162=1129.400,195.226,-63.977,-179.139,9.259,149.576
C05163=1129.404,194.977,-63.952,-179.140,9.256,149.576
C05164=1129.409,194.728,-63.928,-179.142,9.254,149.576
C05165=1129.413,194.480,-63.904,-179.144,9.251,149.575
C05166=1129.418,194.231,-63.880,-179.146,9.249,149.575
C05167=1129.422,193.982,-63.855,-179.147,9.246,149.575
C05168=1129.427,193.733,-63.831,-179.149,9.244,149.575
C05169=1129.432,193.484,-63.807,-179.151,9.241,149.575
C05170=1129.436,193.235,-63.782,-179.152,9.238,149.575
C05171=1129.440,192.987,-63.758,-179.154,9.236,149.574
C05172=1129.445,192.738,-63.733,-179.156,9.233,149.574
C05173=1129.450,192.489,-63.709,-179.158,9.230,149.574
C05174=1129.454,192.240,-63.685,-179.160,9.228,149.574
C05175=1129.459,191.992,-63.660,-179.162,9.225,149.574
C05176=1129.463,191.743,-63.636,-179.163,9.223,149.574
C05177=1129.468,191.494,-63.613,-179.165,9.220,149.574
C05178=1129.473,191.245,-63.588,-179.168,9.217,149.574
C05179=1129.477,190.996,-63.564,-179.169,9.215,149.574
C05180=1129.481,190.748,-63.540,-179.171,9.212,149.574
C05181=1129.486,190.499,-63.516,-179.173,9.209,149.573
C05182=1129.491,190.250,-63.492,-179.175,9.207,149.573
C05183=1129.495,190.001,-63.467,-179.178,9.204,149.573
C05184=1129.499,189.753,-63.443,-179.180,9.201,149.573
C05185=1129.504,189.504,-63.418,-179.182,9.199,149.573
C05186=1129.509,189.255,-63.395,-179.184,9.196,149.573
C05187=1129.513,189.006,-63.371,-179.186,9.194,149.573
C05188=1129.517,188.757,-63.346,-179.189,9.190,149.573
C05189=1129.523,188.508,-63.323,-179.191,9.187,149.573
C05190=1129.527,188.260,-63.298,-179.193,9.185,149.573
C05191=1129.531,188.011,-63.274,-179.196,9.182,149.573
C05192=1129.536,187.762,-63.251,-179.197,9.180,149.573
C05193=1129.540,187.514,-63.227,-179.200,9.176,149.573
C05194=1129.546,187.265,-63.202,-179.202,9.173,149.573
C05195=1129.550,187.015,-63.179,-179.205,9.170,149.573
C05196=1129.554,186.767,-63.154,-179.207,9.168,149.573
C05197=1129.559,186.518,-63.130,-179.209,9.165,149.573
C05198=1129.563,186.269,-63.107,-179.212,9.162,149.573
C05199=1129.568,186.021,-63.083,-179.214,9.159,149.573
C05200=1129.572,185.806,-63.062,-179.217,9.157,149.573
C05201=1129.575,185.592,-63.041,-179.219,9.153,149.573
C05202=1129.580,185.378,-63.021,-179.221,9.151,149.573
C05203=1129.584,185.163,-63.000,-179.223,9.149,149.573
C05204=1129.587,184.949,-62.980,-179.226,9.146,149.573
C05205=1129.591,184.734,-62.959,-179.228,9.143,149.573
C05206=1129.595,184.521,-62.939,-179.230,9.141,149.573
C05207=1129.599,184.306,-62.918,-179.232,9.138,149.573
C05208=1129.604,184.057,-62.895,-179.235,9.135,149.573
C05209=1129.608,183.809,-62.871,-179.237,9.132,149.573
C05210=1129.613,183.560,-62.847,-179.241,9.129,149.573
C05211=1129.618,183.311,-62.824,-179.244,9.125,149.573
C05212=1129.622,183.061,-62.800,-179.246,9.122,149.573
C05213=1129.626,182.812,-62.776,-179.249,9.119,149.573
C05214=1129.631,182.564,-62.752,-179.252,9.117,149.573
C05215=1129.635,182.315,-62.729,-179.255,9.113,149.573
C05216=1129.640,182.066,-62.705,-179.257,9.110,149.573
C05217=1129.645,181.817,-62.681,-179.260,9.107,149.573
C05218=1129.649,181.568,-62.658,-179.263,9.103,149.573
C05219=1129.654,181.319,-62.635,-179.266,9.100,149.573
C05220=1129.658,181.071,-62.611,-179.269,9.096,149.573
C05221=1129.663,180.822,-62.587,-179.272,9.093,149.573
C05222=1129.668,180.573,-62.564,-179.275,9.089,149.573
C05223=1129.672,180.324,-62.541,-179.278,9.087,149.573
C05224=1129.677,180.075,-62.516,-179.281,9.083,149.573
C05225=1129.682,179.826,-62.493,-179.284,9.080,149.573
C05226=1129.686,179.577,-62.470,-179.287,9.076,149.573
C05227=1129.690,179.329,-62.447,-179.291,9.072,149.573
C05228=1129.695,179.080,-62.423,-179.293,9.069,149.573
C05229=1129.699,178.831,-62.400,-179.296,9.066,149.573
C05230=1129.704,178.582,-62.376,-179.297,9.063,149.573
C05231=1129.709,178.333,-62.353,-179.300,9.060,149.573
C05232=1129.713,178.084,-62.329,-179.301,9.058,149.573
C05233=1129.718,177.835,-62.306,-179.304,9.054,149.573
C05234=1129.722,177.586,-62.283,-179.306,9.051,149.573
C05235=1129.727,177.339,-62.260,-179.308,9.049,149.573
C05236=1129.732,177.090,-62.236,-179.310,9.045,149.572
C05237=1129.736,176.841,-62.213,-179.312,9.043,149.572
C05238=1129.741,176.592,-62.190,-179.314,9.040,149.572
C05239=1129.745,176.343,-62.167,-179.317,9.037,149.572
C05240=1129.750,176.094,-62.143,-179.318,9.034,149.572
C05241=1129.755,175.845,-62.120,-179.321,9.031,149.572
C05242=1129.759,175.596,-62.097,-179.323,9.028,149.572
C05243=1129.764,175.347,-62.073,-179.325,9.025,149.572
C05244=1129.768,175.098,-62.051,-179.327,9.022,149.572
C05245=1129.773,174.849,-62.027,-179.330,9.019,149.571
C05246=1129.778,174.601,-62.004,-179.331,9.016,149.571
C05247=1129.783,174.352,-61.981,-179.334,9.013,149.571
C05248=1129.787,174.103,-61.958,-179.337,9.010,149.571
C05249=1129.791,173.854,-61.935,-179.339,9.007,149.571
C05250=1129.796,173.605,-61.911,-179.341,9.004,149.571
C05251=1129.800,173.356,-61.889,-179.343,9.001,149.571
C05252=1129.805,173.106,-61.866,-179.346,8.998,149.571
C05253=1129.810,172.858,-61.843,-179.348,8.995,149.571
C05254=1129.815,172.609,-61.820,-179.350,8.992,149.571
C05255=1129.819,172.360,-61.797,-179.352,8.989,149.571
C05256=1129.823,172.145,-61.777,-179.354,8.987,149.570
C05257=1129.827,171.932,-61.757,-179.356,8.983,149.570
C05258=1129.830,171.717,-61.738,-179.358,8.981,149.570
C05259=1129.835,171.503,-61.717,-179.360,8.979,149.570
C05260=1129.838,171.288,-61.698,-179.362,8.976,149.570
C05261=1129.843,171.073,-61.678,-179.364,8.973,149.570
C05262=1129.846,170.859,-61.658,-179.366,8.971,149.570
C05263=1129.851,170.645,-61.638,-179.368,8.968,149.570
C05264=1129.855,170.396,-61.615,-179.370,8.965,149.570
C05265=1129.860,170.146,-61.593,-179.372,8.962,149.570
C05266=1129.864,169.898,-61.570,-179.375,8.959,149.570
C05267=1129.869,169.649,-61.547,-179.377,8.955,149.570
C05268=1129.873,169.401,-61.524,-179.380,8.952,149.570
C05269=1129.878,169.151,-61.502,-179.381,8.950,149.569
C05270=1129.883,168.902,-61.478,-179.384,8.947,149.569
C05271=1129.888,168.654,-61.456,-179.386,8.943,149.569
C05272=1129.893,168.404,-61.433,-179.389,8.940,149.569
C05273=1129.897,168.155,-61.410,-179.391,8.937,149.569
C05274=1129.901,167.906,-61.387,-179.393,8.934,149.569
C05275=1129.906,167.658,-61.365,-179.396,8.931,149.569
C05276=1129.911,167.409,-61.342,-179.398,8.928,149.569
C05277=1129.915,167.160,-61.319,-179.401,8.924,149.569
C05278=1129.920,166.910,-61.297,-179.403,8.921,149.569
C05279=1129.924,166.662,-61.274,-179.406,8.918,149.569
C05280=1129.929,166.413,-61.252,-179.408,8.915,149.569
C05281=1129.933,166.164,-61.229,-179.411,8.912,149.569
C05282=1129.939,165.915,-61.207,-179.413,8.908,149.568
C05283=1129.943,165.666,-61.184,-179.415,8.905,149.568
C05284=1129.948,165.417,-61.161,-179.418,8.902,149.568
C05285=1129.953,165.169,-61.139,-179.420,8.899,149.568
C05286=1129.958,164.919,-61.116,-179.422,8.895,149.568
C05287=1129.962,164.670,-61.093,-179.425,8.892,149.568
C05288=1129.966,164.422,-61.072,-179.427,8.889,149.568
C05289=1129.971,164.173,-61.048,-179.430,8.886,149.568
C05290=1129.975,163.923,-61.026,-179.432,8.883,149.568
C05291=1129.981,163.675,-61.003,-179.435,8.879,149.568
C05292=1129.985,163.426,-60.981,-179.437,8.876,149.568
C05293=1129.989,163.176,-60.959,-179.440,8.873,149.568
C05294=1129.994,162.928,-60.936,-179.442,8.870,149.567
C05295=1129.999,162.679,-60.914,-179.444,8.867,149.567
C05296=1130.003,162.430,-60.891,-179.447,8.863,149.567
C05297=1130.008,162.181,-60.869,-179.449,8.860,149.567
C05298=1130.013,161.932,-60.847,-179.452,8.856,149.567
C05299=1130.017,161.684,-60.825,-179.455,8.853,149.567
C05300=1130.021,161.434,-60.803,-179.457,8.850,149.567
C05301=1130.026,161.185,-60.780,-179.460,8.847,149.567
C05302=1130.031,160.937,-60.758,-179.462,8.843,149.567
C05303=1130.035,160.687,-60.735,-179.464,8.840,149.567
C05304=1130.041,160.438,-60.713,-179.467,8.836,149.567
C05305=1130.045,160.189,-60.691,-179.470,8.833,149.567
C05306=1130.050,159.941,-60.669,-179.472,8.830,149.566
C05307=1130.054,159.692,-60.647,-179.474,8.827,149.566
C05308=1130.059,159.442,-60.624,-179.477,8.824,149.566
C05309=1130.064,159.193,-60.602,-179.480,8.819,149.566
C05310=1130.068,158.944,-60.580,-179.482,8.816,149.566
C05311=1130.073,158.695,-60.559,-179.485,8.813,149.566
C05312=1130.077,158.481,-60.540,-179.487,8.810,149.566
C05313=1130.081,158.266,-60.520,-179.489,8.806,149.566
C05314=1130.085,158.052,-60.501,-179.491,8.804,149.566
C05315=1130.089,157.837,-60.483,-179.494,8.801,149.566
C05316=1130.092,157.622,-60.463,-179.496,8.798,149.565
C05317=1130.097,157.408,-60.444,-179.498,8.795,149.565
C05318=1130.101,157.194,-60.425,-179.500,8.792,149.565
C05319=1130.105,156.979,-60.407,-179.502,8.789,149.565
C05320=1130.109,156.730,-60.385,-179.505,8.785,149.565
C05321=1130.115,156.481,-60.362,-179.508,8.782,149.565
C05322=1130.119,156.231,-60.340,-179.510,8.778,149.565
C05323=1130.124,155.983,-60.319,-179.513,8.775,149.565
C05324=1130.128,155.733,-60.297,-179.516,8.771,149.565
C05325=1130.133,155.485,-60.275,-179.518,8.768,149.565
C05326=1130.137,155.235,-60.253,-179.520,8.765,149.565
C05327=1130.142,154.987,-60.231,-179.524,8.761,149.565
C05328=1130.147,154.737,-60.209,-179.526,8.757,149.564
C05329=1130.151,154.489,-60.187,-179.529,8.753,149.564
C05330=1130.156,154.240,-60.166,-179.531,8.750,149.564
C05331=1130.161,153.991,-60.144,-179.534,8.746,149.564
C05332=1130.165,153.742,-60.122,-179.536,8.742,149.564
C05333=1130.170,153.493,-60.100,-179.539,8.739,149.564
C05334=1130.175,153.244,-60.078,-179.542,8.735,149.564
C05335=1130.180,152.995,-60.057,-179.545,8.731,149.563
C05336=1130.184,152.746,-60.035,-179.547,8.728,149.563
C05337=1130.189,152.497,-60.014,-179.550,8.724,149.563
C05338=1130.193,152.248,-59.992,-179.552,8.721,149.563
C05339=1130.198,151.999,-59.970,-179.555,8.716,149.563
C05340=1130.203,151.750,-59.949,-179.558,8.713,149.563
C05341=1130.208,151.500,-59.927,-179.560,8.709,149.563
C05342=1130.212,151.252,-59.905,-179.563,8.706,149.563
C05343=1130.217,151.003,-59.883,-179.565,8.702,149.562
C05344=1130.222,150.753,-59.862,-179.569,8.698,149.562
C05345=1130.227,150.505,-59.840,-179.571,8.694,149.562
C05346=1130.232,150.256,-59.819,-179.574,8.690,149.562
C05347=1130.236,150.006,-59.797,-179.577,8.686,149.562
C05348=1130.241,149.757,-59.776,-179.579,8.683,149.562
C05349=1130.245,149.509,-59.755,-179.582,8.679,149.562
C05350=1130.250,149.259,-59.733,-179.585,8.675,149.562
C05351=1130.255,149.010,-59.712,-179.587,8.671,149.561
C05352=1130.260,148.761,-59.691,-179.590,8.667,149.561
C05353=1130.265,148.512,-59.669,-179.593,8.663,149.561
C05354=1130.269,148.263,-59.647,-179.595,8.660,149.561
C05355=1130.273,148.014,-59.627,-179.598,8.656,149.561
C05356=1130.278,147.766,-59.605,-179.601,8.652,149.561
C05357=1130.283,147.516,-59.584,-179.604,8.647,149.560
C05358=1130.288,147.267,-59.562,-179.606,8.644,149.560
C05359=1130.292,147.018,-59.542,-179.609,8.640,149.560
C05360=1130.297,146.769,-59.520,-179.611,8.636,149.560
C05361=1130.302,146.520,-59.499,-179.615,8.632,149.560
C05362=1130.306,146.271,-59.477,-179.617,8.628,149.560
C05363=1130.311,146.022,-59.456,-179.620,8.623,149.559
C05364=1130.316,145.773,-59.435,-179.623,8.620,149.559
C05365=1130.321,145.524,-59.414,-179.625,8.616,149.559
C05366=1130.326,145.275,-59.393,-179.628,8.612,149.559
C05367=1130.330,145.026,-59.371,-179.631,8.608,149.559
C05368=1130.334,144.811,-59.353,-179.632,8.605,149.558
C05369=1130.338,144.596,-59.335,-179.634,8.602,149.558
C05370=1130.342,144.381,-59.317,-179.635,8.599,149.558
C05371=1130.346,144.167,-59.298,-179.636,8.596,149.558
C05372=1130.350,143.952,-59.281,-179.637,8.593,149.557
C05373=1130.354,143.737,-59.262,-179.639,8.590,149.557
C05374=1130.358,143.523,-59.245,-179.640,8.587,149.556
C05375=1130.362,143.308,-59.226,-179.640,8.585,149.556
C05376=1130.367,143.059,-59.206,-179.642,8.581,149.556
C05377=1130.372,142.810,-59.185,-179.643,8.579,149.556
C05378=1130.377,142.561,-59.163,-179.645,8.575,149.555
C05379=1130.381,142.312,-59.142,-179.646,8.572,149.555
C05380=1130.386,142.062,-59.121,-179.648,8.568,149.555
C05381=1130.390,141.813,-59.101,-179.649,8.565,149.554
C05382=1130.395,141.565,-59.079,-179.651,8.563,149.554
C05383=1130.400,141.315,-59.058,-179.652,8.559,149.553
C05384=1130.405,141.066,-59.038,-179.653,8.556,149.553
C05385=1130.410,140.817,-59.017,-179.655,8.552,149.553
C05386=1130.415,140.568,-58.997,-179.656,8.549,149.552
C05387=1130.419,140.319,-58.975,-179.658,8.546,149.552
C05388=1130.423,140.070,-58.954,-179.659,8.542,149.552
C05389=1130.428,139.821,-58.933,-179.662,8.539,149.551
C05390=1130.433,139.572,-58.913,-179.663,8.536,149.551
C05391=1130.438,139.323,-58.892,-179.665,8.532,149.551
C05392=1130.442,139.074,-58.872,-179.666,8.529,149.550
C05393=1130.447,138.825,-58.850,-179.668,8.526,149.550
C05394=1130.452,138.576,-58.830,-179.669,8.523,149.550
C05395=1130.457,138.327,-58.809,-179.671,8.519,149.549
C05396=1130.461,138.078,-58.788,-179.672,8.516,149.549
C05397=1130.467,137.829,-58.767,-179.673,8.513,149.549
C05398=1130.471,137.580,-58.747,-179.675,8.510,149.548
C05399=1130.476,137.330,-58.726,-179.676,8.507,149.548
C05400=1130.480,137.081,-58.705,-179.678,8.503,149.548
C05401=1130.485,136.831,-58.684,-179.679,8.500,149.548
C05402=1130.490,136.582,-58.664,-179.681,8.496,149.547
C05403=1130.495,136.333,-58.643,-179.683,8.494,149.547
C05404=1130.499,136.084,-58.623,-179.684,8.490,149.546
C05405=1130.504,135.835,-58.602,-179.686,8.486,149.546
C05406=1130.509,135.586,-58.581,-179.688,8.484,149.546
C05407=1130.513,135.337,-58.561,-179.689,8.480,149.546
C05408=1130.518,135.088,-58.540,-179.691,8.477,149.545
C05409=1130.523,134.839,-58.519,-179.692,8.473,149.545
C05410=1130.527,134.590,-58.499,-179.694,8.470,149.545
C05411=1130.532,134.341,-58.478,-179.696,8.467,149.544
C05412=1130.537,134.092,-58.458,-179.697,8.464,149.544
C05413=1130.542,133.842,-58.437,-179.699,8.460,149.544
C05414=1130.547,133.593,-58.416,-179.700,8.458,149.544
C05415=1130.551,133.345,-58.396,-179.702,8.454,149.543
C05416=1130.556,133.095,-58.376,-179.704,8.451,149.543
C05417=1130.561,132.846,-58.355,-179.705,8.447,149.542
C05418=1130.565,132.597,-58.335,-179.707,8.444,149.542
C05419=1130.570,132.348,-58.314,-179.709,8.441,149.542
C05420=1130.575,132.099,-58.294,-179.710,8.437,149.542
C05421=1130.579,131.850,-58.273,-179.712,8.434,149.541
C05422=1130.585,131.600,-58.253,-179.714,8.431,149.541
C05423=1130.590,131.351,-58.233,-179.715,8.427,149.541
C05424=1130.594,131.137,-58.215,-179.717,8.424,149.540
C05425=1130.597,130.922,-58.198,-179.718,8.422,149.540
C05426=1130.602,130.707,-58.180,-179.720,8.419,149.540
C05427=1130.606,130.492,-58.163,-179.721,8.416,149.540
C05428=1130.610,130.277,-58.145,-179.723,8.413,149.540
C05429=1130.614,130.062,-58.127,-179.724,8.411,149.539
C05430=1130.618,129.848,-58.110,-179.726,8.408,149.539
C05431=1130.622,129.633,-58.093,-179.727,8.405,149.539
C05432=1130.627,129.384,-58.073,-179.729,8.401,149.539
C05433=1130.632,129.135,-58.052,-179.731,8.398,149.538
C05434=1130.637,128.885,-58.032,-179.732,8.395,149.538
C05435=1130.641,128.636,-58.012,-179.734,8.391,149.538
C05436=1130.646,128.387,-57.991,-179.736,8.388,149.537
C05437=1130.650,128.138,-57.971,-179.737,8.385,149.537
C05438=1130.656,127.889,-57.951,-179.739,8.382,149.537
C05439=1130.661,127.640,-57.931,-179.741,8.378,149.537
C05440=1130.665,127.391,-57.911,-179.742,8.375,149.536
C05441=1130.670,127.142,-57.891,-179.745,8.372,149.536
C05442=1130.674,126.893,-57.870,-179.747,8.368,149.536
C05443=1130.680,126.643,-57.850,-179.748,8.365,149.535
C05444=1130.684,126.394,-57.830,-179.750,8.361,149.535
C05445=1130.689,126.145,-57.810,-179.752,8.358,149.535
C05446=1130.694,125.896,-57.790,-179.753,8.355,149.535
C05447=1130.698,125.647,-57.769,-179.755,8.351,149.534
C05448=1130.703,125.398,-57.750,-179.757,8.348,149.534
C05449=1130.708,125.149,-57.729,-179.758,8.345,149.534
